// ============================================
// DB_RecipeProgram2 - Program 2
// Lines: 500
// CHUNKS: 5 x 100
// Generated by SpinningCam  [2026-09-29 00:03:31]
// !!! CONTINUOUS MOTION (CMD=2) - EXPERIMENTAL PLC ONLY !!!
// Load ONLY on the continuous-motion PLC build. A production PLC
// skips CMD=2 lines and jumps straight between the other points.
// T=0.045 s, corner tol=0.2 mm, F min=180, exact stop at >= 90 deg, stop slow-down=OFF
// CMD=2 lines: 385, exact corners: 39, slowed corners: 36 (+57 leaving), slowed stops: 0
// ============================================
//
// --- MAKINE AYARLARI ---
// Machine Origin  : X=0.0, Z=0.0
// Axis Direction  : X=NORMAL, Z=NORMAL
// Output Mode     : RADIUS
// G54 Offset      : X=0.0, Z=0.0
// Home            : X=-394.0, Z=-174.0
// Retract         : X=-10.0, Z=-10.0
//
// --- PARCA / BLANK ---
// Blank Radius    : 77.8 mm
// Blank Z Shift   : 0.0 mm
// Final Thickness : 0.8 mm
// Min Safety Gap  : 0.0 mm
//
// --- MANDREL POZISYON ---
// Mandrel Offset  : X=0.0, Z=0.0
// Mandrel Rot     : Rx=90.0, Ry=0.0, Rz=0.0
//
// --- OPERASYONLAR ---
// Op1: ROUGHING, 1 paso, T004, R=44.56mm, RPM=600.0, mm_min=900.0
// Op2: ROUGHING, 1 paso, T004, R=44.56mm, RPM=600.0, mm_min=900.0
// Op3: ROUGHING, 1 paso, T004, R=44.56mm, RPM=600.0, mm_min=900.0
// Op4: ROUGHING, 1 paso, T004, R=44.56mm, RPM=600.0, mm_min=900.0
// Op5: ROUGHING, 1 paso, T004, R=44.56mm, RPM=600.0, mm_min=900.0
// Op6: ROUGHING, 1 paso, T004, R=44.56mm, RPM=600.0, mm_min=800.0
// Op7: ROUGHING, 1 paso, T004, R=44.56mm, RPM=600.0, mm_min=800.0
// Op8: ROUGHING, 1 paso, T004, R=44.56mm, RPM=600.0, mm_min=800.0
// Op9: ROUGHING, 1 paso, T004, R=44.56mm, RPM=600.0, mm_min=800.0
// Op10: ROUGHING, 1 paso, T004, R=44.56mm, RPM=600.0, mm_min=800.0
// Op11: ROUGHING, 1 paso, T004, R=44.56mm, RPM=600.0, mm_min=800.0
// Op12: ROUGHING, 1 paso, T004, R=44.56mm, RPM=600.0, mm_min=800.0
// Op13: ROUGHING, 1 paso, T004, R=44.56mm, RPM=600.0, mm_min=1000.0
// Op14: ROUGHING, 1 paso, T004, R=44.56mm, RPM=600.0, mm_min=1000.0
// Op15: ROUGHING, 1 paso, T004, R=44.56mm, RPM=600.0, mm_min=1000.0
// Op16: ROUGHING, 1 paso, T004, R=44.56mm, RPM=600.0, mm_min=1000.0
// Op17: ROUGHING, 1 paso, T004, R=44.56mm, RPM=600.0, mm_min=1000.0
// Op18: ROUGHING, 1 paso, T004, R=44.56mm, RPM=600.0, mm_min=1000.0
// Op19: ROUGHING, 1 paso, T004, R=44.56mm, RPM=600.0, mm_min=1000.0
// Op20: ROUGHING, 1 paso, T004, R=44.56mm, RPM=600.0, mm_min=1000.0
// Op21: ROUGHING, 1 paso, T004, R=44.56mm, RPM=600.0, mm_min=1000.0
// Op22: ROUGHING, 1 paso, T004, R=44.56mm, RPM=600.0, mm_min=1000.0
// Op23: ROUGHING, 1 paso, T004, R=44.56mm, RPM=600.0, mm_min=1000.0
// Op24: ROUGHING, 1 paso, T004, R=44.56mm, RPM=600.0, mm_min=1000.0
// Op25: ROUGHING, 1 paso, T004, R=44.56mm, RPM=600.0, mm_min=1000.0
// Op26: ROUGHING, 1 paso, T004, R=44.56mm, RPM=600.0, mm_min=1000.0
// Op27: CUTTING, 1 paso, T006, R=20.0mm, RPM=500.0, mm_min=10.0
// Op28: ROUGHING, 1 paso, T004, R=44.56mm, RPM=600.0, mm_min=1000.0
// Op29: ROUGHING, 1 paso, T004, R=44.56mm, RPM=600.0, mm_min=1000.0
// Op30: ROUGHING, 1 paso, T004, R=44.56mm, RPM=600.0, mm_min=1000.0
// Op31: ROUGHING, 1 paso, T004, R=44.56mm, RPM=600.0, mm_min=1000.0
// Op32: ROUGHING, 1 paso, T004, R=44.56mm, RPM=600.0, mm_min=1000.0
// Op33: ROUGHING, 1 paso, T004, R=44.56mm, RPM=600.0, mm_min=1000.0
// Op34: ROUGHING, 1 paso, T004, R=44.56mm, RPM=600.0, mm_min=1000.0
// Op35: ROUGHING, 1 paso, T004, R=44.56mm, RPM=600.0, mm_min=1000.0
// Op36: ROUGHING, 1 paso, T004, R=44.56mm, RPM=600.0, mm_min=1500.0
// Op37: ROUGHING, 1 paso, T004, R=44.56mm, RPM=600.0, mm_min=1500.0
// Op38: ROUGHING, 1 paso, T004, R=44.56mm, RPM=600.0, mm_min=1500.0
// Op39: ROUGHING, 1 paso, T004, R=44.56mm, RPM=600.0, mm_min=1500.0
// Op40: ROUGHING, 1 paso, T004, R=44.56mm, RPM=600.0, mm_min=1500.0
// Op41: ROUGHING, 1 paso, T004, R=44.56mm, RPM=600.0, mm_min=1500.0
// Op42: ROUGHING, 1 paso, T004, R=44.56mm, RPM=600.0, mm_min=1500.0
// Op43: ROUGHING, 1 paso, T004, R=44.56mm, RPM=600.0, mm_min=1500.0
// Op44: ROUGHING, 1 paso, T004, R=44.56mm, RPM=600.0, mm_min=1500.0
// Op45: ROUGHING, 1 paso, T004, R=44.56mm, RPM=600.0, mm_min=1500.0
// Op46: ROUGHING, 1 paso, T004, R=44.56mm, RPM=600.0, mm_min=1500.0
// Op47: ROUGHING, 1 paso, T004, R=44.56mm, RPM=600.0, mm_min=1500.0
// Op48: ROUGHING, 1 paso, T004, R=44.56mm, RPM=600.0, mm_min=1500.0
// Op49: ROUGHING, 1 paso, T004, R=44.56mm, RPM=600.0, mm_min=1500.0
// Op50: ROUGHING, 1 paso, T004, R=44.56mm, RPM=600.0, mm_min=1500.0
// Op51: ROUGHING, 1 paso, T004, R=44.56mm, RPM=600.0, mm_min=1500.0
// Op52: ROUGHING, 1 paso, T004, R=44.56mm, RPM=600.0, mm_min=1500.0
// Op53: ROUGHING, 1 paso, T004, R=44.56mm, RPM=600.0, mm_min=1500.0
// Op54: ROUGHING, 1 paso, T004, R=44.56mm, RPM=600.0, mm_min=1500.0
// Op55: ROUGHING, 1 paso, T004, R=44.56mm, RPM=600.0, mm_min=1500.0
// Op56: ROUGHING, 1 paso, T004, R=44.56mm, RPM=600.0, mm_min=1500.0
// Op57: ROUGHING, 1 paso, T004, R=44.56mm, RPM=600.0, mm_min=1500.0
// Op58: ROUGHING, 1 paso, T004, R=44.56mm, RPM=600.0, mm_min=1500.0
// Op59: ROUGHING, 1 paso, T004, R=44.56mm, RPM=600.0, mm_min=1500.0
// Op60: ROUGHING, 1 paso, T004, R=44.56mm, RPM=800.0, mm_min=1500.0
// Op61: ROUGHING, 1 paso, T004, R=44.56mm, RPM=800.0, mm_min=800.0
// Op62: ROUGHING, 1 paso, T004, R=44.56mm, RPM=800.0, mm_min=800.0
// Op63: ROUGHING, 1 paso, T004, R=44.56mm, RPM=600.0, mm_min=1500.0
// Op64: ROUGHING, 1 paso, T004, R=44.56mm, RPM=600.0, mm_min=1500.0
// Op65: ROUGHING, 1 paso, T004, R=44.56mm, RPM=600.0, mm_min=1500.0
// Op66: ROUGHING, 1 paso, T004, R=44.56mm, RPM=600.0, mm_min=1500.0
// Op67: ROUGHING, 1 paso, T004, R=44.56mm, RPM=600.0, mm_min=1500.0
// Op68: ROUGHING, 1 paso, T004, R=44.56mm, RPM=600.0, mm_min=1500.0
// Op69: ROUGHING, 1 paso, T004, R=44.56mm, RPM=600.0, mm_min=1500.0
// Op70: ROUGHING, 1 paso, T004, R=44.56mm, RPM=600.0, mm_min=1500.0
// Op71: ROUGHING, 1 paso, T004, R=44.56mm, RPM=600.0, mm_min=1500.0
// Op72: ROUGHING, 1 paso, T004, R=44.56mm, RPM=600.0, mm_min=1000.0
// Op73: ROUGHING, 1 paso, T004, R=44.56mm, RPM=600.0, mm_min=1000.0
// Op74: ROUGHING, 1 paso, T004, R=44.56mm, RPM=600.0, mm_min=1000.0
// Op75: ROUGHING, 1 paso, T004, R=44.56mm, RPM=600.0, mm_min=1000.0
// Op76: ROUGHING, 1 paso, T004, R=44.56mm, RPM=600.0, mm_min=1500.0
// Op77: ROUGHING, 1 paso, T004, R=44.56mm, RPM=600.0, mm_min=1000.0
// Op78: ROUGHING, 1 paso, T004, R=44.56mm, RPM=600.0, mm_min=1000.0
// Op79: ROUGHING, 1 paso, T004, R=44.56mm, RPM=600.0, mm_min=1000.0
// Op80: ROUGHING, 1 paso, T004, R=44.56mm, RPM=600.0, mm_min=1000.0
// Op81: ROUGHING, 1 paso, T004, R=44.56mm, RPM=600.0, mm_min=1000.0
// Op82: ROUGHING, 1 paso, T004, R=44.56mm, RPM=600.0, mm_min=1000.0
// Op83: ROUGHING, 1 paso, T004, R=44.56mm, RPM=600.0, mm_min=1000.0
// Op84: ROUGHING, 1 paso, T004, R=44.56mm, RPM=600.0, mm_min=1000.0
// Op85: ROUGHING, 1 paso, T004, R=44.56mm, RPM=600.0, mm_min=1000.0
// Op86: ROUGHING, 1 paso, T004, R=44.56mm, RPM=600.0, mm_min=1000.0
// Op87: ROUGHING, 1 paso, T004, R=44.56mm, RPM=600.0, mm_min=1000.0
// Op88: ROUGHING, 1 paso, T004, R=44.56mm, RPM=600.0, mm_min=1000.0
// Op89: ROUGHING, 1 paso, T004, R=44.56mm, RPM=600.0, mm_min=1000.0
// Op90: ROUGHING, 1 paso, T004, R=44.56mm, RPM=600.0, mm_min=1000.0
// Op91: ROUGHING, 1 paso, T004, R=44.56mm, RPM=600.0, mm_min=1000.0
// Op92: ROUGHING, 1 paso, T004, R=44.56mm, RPM=600.0, mm_min=1000.0
// Op93: ROUGHING, 1 paso, T004, R=44.56mm, RPM=600.0, mm_min=1000.0
// Op94: ROUGHING, 1 paso, T004, R=44.56mm, RPM=600.0, mm_min=1000.0
// Op95: ROUGHING, 1 paso, T004, R=44.56mm, RPM=600.0, mm_min=1000.0
// Op96: ROUGHING, 1 paso, T004, R=44.56mm, RPM=600.0, mm_min=1000.0
// Op97: ROUGHING, 1 paso, T004, R=44.56mm, RPM=600.0, mm_min=1000.0
// Op98: ROUGHING, 1 paso, T004, R=44.56mm, RPM=600.0, mm_min=1000.0
// Op99: ROUGHING, 1 paso, T004, R=44.56mm, RPM=600.0, mm_min=1000.0
// Op100: ROUGHING, 1 paso, T004, R=44.56mm, RPM=600.0, mm_min=1000.0
// Op101: ROUGHING, 1 paso, T004, R=44.56mm, RPM=600.0, mm_min=1000.0
// Op102: ROUGHING, 1 paso, T004, R=44.56mm, RPM=600.0, mm_min=1000.0
// Op103: ROUGHING, 1 paso, T004, R=44.56mm, RPM=600.0, mm_min=1000.0
// Op104: ROUGHING, 1 paso, T004, R=44.56mm, RPM=600.0, mm_min=1000.0
// Op105: ROUGHING, 1 paso, T004, R=44.56mm, RPM=600.0, mm_min=1000.0
// Op106: ROUGHING, 1 paso, T004, R=44.56mm, RPM=600.0, mm_min=1000.0
// Op107: ROUGHING, 1 paso, T004, R=44.56mm, RPM=600.0, mm_min=1000.0
// Op108: ROUGHING, 1 paso, T004, R=44.56mm, RPM=600.0, mm_min=1000.0
// Op109: ROUGHING, 1 paso, T004, R=44.56mm, RPM=600.0, mm_min=1000.0
// Op110: ROUGHING, 1 paso, T004, R=44.56mm, RPM=600.0, mm_min=1000.0
// Op111: ROUGHING, 1 paso, T004, R=44.56mm, RPM=600.0, mm_min=1000.0
// Op112: ROUGHING, 1 paso, T004, R=44.56mm, RPM=600.0, mm_min=1000.0
// Op113: ROUGHING, 1 paso, T004, R=44.56mm, RPM=600.0, mm_min=1000.0
// Op114: ROUGHING, 1 paso, T004, R=44.56mm, RPM=600.0, mm_min=1000.0
// Op115: ROUGHING, 1 paso, T004, R=44.56mm, RPM=600.0, mm_min=1000.0
// Op116: ROUGHING, 1 paso, T004, R=44.56mm, RPM=600.0, mm_min=1000.0
// Op117: ROUGHING, 1 paso, T004, R=44.56mm, RPM=600.0, mm_min=1000.0
// Op118: ROUGHING, 1 paso, T004, R=44.56mm, RPM=600.0, mm_min=1000.0
// Op119: ROUGHING, 1 paso, T004, R=44.56mm, RPM=600.0, mm_min=1000.0
// Op120: ROUGHING, 1 paso, T004, R=44.56mm, RPM=600.0, mm_min=1000.0
// Op121: ROUGHING, 1 paso, T004, R=44.56mm, RPM=600.0, mm_min=1000.0
// Op122: ROUGHING, 1 paso, T004, R=44.56mm, RPM=600.0, mm_min=1000.0
// Op123: ROUGHING, 1 paso, T004, R=44.56mm, RPM=600.0, mm_min=1000.0
// Op124: ROUGHING, 1 paso, T004, R=44.56mm, RPM=600.0, mm_min=1000.0
// Op125: ROUGHING, 1 paso, T004, R=44.56mm, RPM=600.0, mm_min=1000.0
// Op126: ROUGHING, 1 paso, T004, R=44.56mm, RPM=600.0, mm_min=1000.0
// Op127: ROUGHING, 1 paso, T004, R=44.56mm, RPM=600.0, mm_min=1000.0
// Op128: ROUGHING, 1 paso, T004, R=44.56mm, RPM=600.0, mm_min=1000.0
// Op129: CUTTING, 1 paso, T006, R=20.0mm, RPM=500.0, mm_min=7.0
// Op130: ROUGHING, 1 paso, T004, R=44.56mm, RPM=600.0, mm_min=1000.0
// Op131: ROUGHING, 1 paso, T004, R=44.56mm, RPM=600.0, mm_min=1000.0
// Op132: ROUGHING, 1 paso, T004, R=44.56mm, RPM=600.0, mm_min=1000.0
// Op133: ROUGHING, 1 paso, T004, R=44.56mm, RPM=600.0, mm_min=1000.0
// Op134: ROUGHING, 1 paso, T004, R=44.56mm, RPM=600.0, mm_min=1000.0
// Op135: ROUGHING, 1 paso, T004, R=44.56mm, RPM=600.0, mm_min=1000.0
// Op136: ROUGHING, 1 paso, T004, R=44.56mm, RPM=600.0, mm_min=1000.0
// Op137: ROUGHING, 1 paso, T004, R=44.56mm, RPM=600.0, mm_min=400.0
// Op138: ROUGHING, 1 paso, T004, R=44.56mm, RPM=600.0, mm_min=400.0
// Op139: ROUGHING, 1 paso, T004, R=44.56mm, RPM=600.0, mm_min=400.0
// Op140: ROUGHING, 1 paso, T004, R=44.56mm, RPM=600.0, mm_min=1000.0
// Op141: ROUGHING, 1 paso, T004, R=44.56mm, RPM=600.0, mm_min=400.0
// Op142: ROUGHING, 1 paso, T004, R=44.56mm, RPM=600.0, mm_min=400.0
// Op143: ROUGHING, 1 paso, T004, R=44.56mm, RPM=600.0, mm_min=400.0
// Op144: ROUGHING, 1 paso, T004, R=44.56mm, RPM=600.0, mm_min=400.0
// Op145: ROUGHING, 1 paso, T004, R=44.56mm, RPM=600.0, mm_min=400.0
// Op146: ROUGHING, 1 paso, T004, R=44.56mm, RPM=600.0, mm_min=400.0
// Op147: ROUGHING, 1 paso, T004, R=44.56mm, RPM=600.0, mm_min=400.0
// Op148: ROUGHING, 1 paso, T004, R=44.56mm, RPM=600.0, mm_min=400.0
// Op149: ROUGHING, 1 paso, T004, R=44.56mm, RPM=600.0, mm_min=400.0
// Op150: ROUGHING, 1 paso, T004, R=44.56mm, RPM=600.0, mm_min=400.0
// Op151: ROUGHING, 1 paso, T004, R=44.56mm, RPM=600.0, mm_min=400.0
// Op152: ROUGHING, 1 paso, T004, R=44.56mm, RPM=600.0, mm_min=400.0
// Op153: ROUGHING, 1 paso, T004, R=44.56mm, RPM=600.0, mm_min=400.0
// Op154: ROUGHING, 1 paso, T004, R=44.56mm, RPM=600.0, mm_min=400.0
// Op155: ROUGHING, 1 paso, T004, R=44.56mm, RPM=600.0, mm_min=400.0
// Op156: ROUGHING, 1 paso, T004, R=44.56mm, RPM=600.0, mm_min=400.0
// Op157: ROUGHING, 1 paso, T004, R=44.56mm, RPM=600.0, mm_min=400.0
// Op158: ROUGHING, 1 paso, T004, R=44.56mm, RPM=600.0, mm_min=400.0
// Op159: ROUGHING, 1 paso, T004, R=44.56mm, RPM=600.0, mm_min=400.0
// Op160: ROUGHING, 1 paso, T004, R=44.56mm, RPM=600.0, mm_min=400.0
// Op161: ROUGHING, 1 paso, T004, R=44.56mm, RPM=600.0, mm_min=400.0
// Op162: ROUGHING, 1 paso, T004, R=44.56mm, RPM=600.0, mm_min=400.0
// Op163: ROUGHING, 1 paso, T004, R=44.56mm, RPM=600.0, mm_min=400.0
// Op164: ROUGHING, 1 paso, T004, R=44.56mm, RPM=600.0, mm_min=400.0
// Op165: ROUGHING, 1 paso, T004, R=44.56mm, RPM=600.0, mm_min=400.0
// Op166: ROUGHING, 1 paso, T004, R=44.56mm, RPM=600.0, mm_min=400.0
// Op167: ROUGHING, 1 paso, T004, R=44.56mm, RPM=800.0, mm_min=400.0
// Op168: ROUGHING, 1 paso, T004, R=44.56mm, RPM=800.0, mm_min=400.0
// Op169: ROUGHING, 1 paso, T004, R=44.56mm, RPM=800.0, mm_min=400.0
// Op170: ROUGHING, 1 paso, T004, R=44.56mm, RPM=800.0, mm_min=400.0
// Op171: ROUGHING, 1 paso, T004, R=44.56mm, RPM=800.0, mm_min=400.0
// Op172: ROUGHING, 1 paso, T004, R=44.56mm, RPM=800.0, mm_min=400.0
// Op173: ROUGHING, 1 paso, T004, R=44.56mm, RPM=800.0, mm_min=400.0
// Op174: ROUGHING, 1 paso, T004, R=44.56mm, RPM=800.0, mm_min=400.0
// Op175: ROUGHING, 1 paso, T004, R=44.56mm, RPM=800.0, mm_min=400.0
// Op176: ROUGHING, 1 paso, T004, R=44.56mm, RPM=800.0, mm_min=400.0
// Op177: ROUGHING, 1 paso, T004, R=44.56mm, RPM=800.0, mm_min=400.0
// Op178: ROUGHING, 1 paso, T004, R=44.56mm, RPM=800.0, mm_min=400.0
// Op179: ROUGHING, 1 paso, T004, R=44.56mm, RPM=800.0, mm_min=400.0
// Op180: ROUGHING, 1 paso, T004, R=44.56mm, RPM=800.0, mm_min=400.0
// Op181: ROUGHING, 1 paso, T004, R=44.56mm, RPM=800.0, mm_min=400.0
// Op182: ROUGHING, 1 paso, T004, R=44.56mm, RPM=800.0, mm_min=400.0
// Op183: ROUGHING, 1 paso, T004, R=44.56mm, RPM=800.0, mm_min=400.0
// ============================================

DATA_BLOCK "DB_RecipeProgram2"
{ S7_Optimized_Access := 'FALSE' }
VERSION : 0.2
UNLINKED
NON_RETAIN
    VAR
        Header : "RecipeHeader";
        Lines1 : Array[0..99] of "RecipeLine";  // global lines 0..99
        Lines2 : Array[0..99] of "RecipeLine";  // global lines 100..199
        Lines3 : Array[0..99] of "RecipeLine";  // global lines 200..299
        Lines4 : Array[0..99] of "RecipeLine";  // global lines 300..399
        Lines5 : Array[0..99] of "RecipeLine";  // global lines 400..499
    END_VAR
BEGIN
    // Header
    Header.sName := 'Program 2';
    Header.LineCount := 500;
    Header.Valid := TRUE;
    Header.PreScanned := FALSE;
    Header.MinX := 0.000;
    Header.MaxX := 273.391;
    Header.MinZ := 0.000;
    Header.MaxZ := 344.140;

    // --- Tool table (CAM-authored) ---
    Header.ProvidesToolConfig := TRUE;
    Header.ToolCount := 4;
    Header.AutoCalcAngles := FALSE;
    Header.ToolCode_List[1] := 4;
    Header.ToolCode_List[2] := 5;
    Header.ToolCode_List[3] := 6;
    Header.ToolCode_List[4] := 7;
    Header.ToolAngle_List[1] := 0.0;
    Header.ToolAngle_List[2] := 120.0;
    Header.ToolAngle_List[3] := 240.0;
    Header.ToolAngle_List[4] := 360.0;

    // --- Integrity ---
    // Order-sensitive sum over CMD+Param+F of lines 0..LineCount-1.
    // The PLC recomputes it after reassembling the chunks and refuses
    // to run on a mismatch (16#0316). X/Z are excluded on purpose:
    // float32-vs-float64 rounding would eventually cry wolf.
    Header.ProvidesChecksum := TRUE;
    Header.Checksum := 106433390;

    // Recipe Lines (500 total)

    // --- Lines1 (global lines 0..99) ---
    Lines1[0].X := 0.000; Lines1[0].Z := 0.000; Lines1[0].F := 0; Lines1[0].CMD := 40; Lines1[0].Param := 80; // Cylinder GOTO P80
    Lines1[1].X := 0.000; Lines1[1].Z := 0.000; Lines1[1].F := 0; Lines1[1].CMD := 10; Lines1[1].Param := 4; // Tool Change T4
    Lines1[2].X := 0.000; Lines1[2].Z := 0.000; Lines1[2].F := 0; Lines1[2].CMD := 20; Lines1[2].Param := 60; // Spindle ON 600 RPM
    Lines1[3].X := 0.000; Lines1[3].Z := 0.000; Lines1[3].F := 0; Lines1[3].CMD := 41; Lines1[3].Param := 1; // M41 (Clamp On) P1 [Op1 P1]
    Lines1[4].X := 272.912; Lines1[4].Z := 176.000; Lines1[4].F := 0; Lines1[4].CMD := 0; Lines1[4].Param := 0; // G0 Rapid [Op1 P1]
    Lines1[5].X := 272.901; Lines1[5].Z := 181.258; Lines1[5].F := 736; Lines1[5].CMD := 2; Lines1[5].Param := 0; // G1 Continuous [Op1 P1]
    Lines1[6].X := 272.111; Lines1[6].Z := 183.280; Lines1[6].F := 395; Lines1[6].CMD := 2; Lines1[6].Param := 0; // G1 Continuous [Op1 P1]
    Lines1[7].X := 270.164; Lines1[7].Z := 184.240; Lines1[7].F := 395; Lines1[7].CMD := 2; Lines1[7].Param := 0; // G1 Continuous [Op1 P1]
    Lines1[8].X := 178.498; Lines1[8].Z := 192.302; Lines1[8].F := 736; Lines1[8].CMD := 2; Lines1[8].Param := 0; // G1 Continuous [Op1 P1]
    Lines1[9].X := 173.498; Lines1[9].Z := 187.302; Lines1[9].F := 0; Lines1[9].CMD := 0; Lines1[9].Param := 0; // G0 Rapid [Op1 P1]
    Lines1[10].X := 173.498; Lines1[10].Z := 187.302; Lines1[10].F := 0; Lines1[10].CMD := 41; Lines1[10].Param := 2; // M41 (Clamp On) P2 [Op2 P1]
    Lines1[11].X := 273.001; Lines1[11].Z := 182.538; Lines1[11].F := 0; Lines1[11].CMD := 0; Lines1[11].Param := 0; // G0 Rapid [Op2 P1]
    Lines1[12].X := 272.998; Lines1[12].Z := 183.142; Lines1[12].F := 866; Lines1[12].CMD := 2; Lines1[12].Param := 0; // G1 Continuous [Op2 P1]
    Lines1[13].X := 272.418; Lines1[13].Z := 184.905; Lines1[13].F := 426; Lines1[13].CMD := 2; Lines1[13].Param := 0; // G1 Continuous [Op2 P1]
    Lines1[14].X := 270.650; Lines1[14].Z := 186.059; Lines1[14].F := 426; Lines1[14].CMD := 2; Lines1[14].Param := 0; // G1 Continuous [Op2 P1]
    Lines1[15].X := 180.388; Lines1[15].Z := 206.156; Lines1[15].F := 758; Lines1[15].CMD := 2; Lines1[15].Param := 0; // G1 Continuous [Op2 P1]
    Lines1[16].X := 272.995; Lines1[16].Z := 184.077; Lines1[16].F := 0; Lines1[16].CMD := 0; Lines1[16].Param := 0; // G0 Rapid [Op3 P1]
    Lines1[17].X := 272.992; Lines1[17].Z := 184.868; Lines1[17].F := 449; Lines1[17].CMD := 2; Lines1[17].Param := 0; // G1 Continuous [Op3 P1]
    Lines1[18].X := 270.873; Lines1[18].Z := 187.725; Lines1[18].F := 449; Lines1[18].CMD := 2; Lines1[18].Param := 0; // G1 Continuous [Op3 P1]
    Lines1[19].X := 182.286; Lines1[19].Z := 214.928; Lines1[19].F := 449; Lines1[19].CMD := 2; Lines1[19].Param := 0; // G1 Continuous [Op3 P1]
    Lines1[20].X := 273.006; Lines1[20].Z := 181.000; Lines1[20].F := 0; Lines1[20].CMD := 0; Lines1[20].Param := 0; // G0 Rapid [Op4 P1]
    Lines1[21].X := 272.984; Lines1[21].Z := 186.988; Lines1[21].F := 478; Lines1[21].CMD := 2; Lines1[21].Param := 0; // G1 Continuous [Op4 P1]
    Lines1[22].X := 271.113; Lines1[22].Z := 189.757; Lines1[22].F := 478; Lines1[22].CMD := 2; Lines1[22].Param := 0; // G1 Continuous [Op4 P1]
    Lines1[23].X := 185.053; Lines1[23].Z := 224.685; Lines1[23].F := 478; Lines1[23].CMD := 2; Lines1[23].Param := 0; // G1 Continuous [Op4 P1]
    Lines1[24].X := 273.006; Lines1[24].Z := 181.000; Lines1[24].F := 0; Lines1[24].CMD := 0; Lines1[24].Param := 0; // G0 Rapid [Op5 P1]
    Lines1[25].X := 272.980; Lines1[25].Z := 188.100; Lines1[25].F := 498; Lines1[25].CMD := 2; Lines1[25].Param := 0; // G1 Continuous [Op5 P1]
    Lines1[26].X := 271.253; Lines1[26].Z := 190.806; Lines1[26].F := 498; Lines1[26].CMD := 2; Lines1[26].Param := 0; // G1 Continuous [Op5 P1]
    Lines1[27].X := 187.038; Lines1[27].Z := 230.259; Lines1[27].F := 498; Lines1[27].CMD := 2; Lines1[27].Param := 0; // G1 Continuous [Op5 P1]
    Lines1[28].X := 273.106; Lines1[28].Z := 181.000; Lines1[28].F := 0; Lines1[28].CMD := 0; Lines1[28].Param := 0; // G0 Rapid [Op6 P1]
    Lines1[29].X := 273.076; Lines1[29].Z := 189.172; Lines1[29].F := 512; Lines1[29].CMD := 2; Lines1[29].Param := 0; // G1 Continuous [Op6 P1]
    Lines1[30].X := 271.442; Lines1[30].Z := 191.832; Lines1[30].F := 512; Lines1[30].CMD := 2; Lines1[30].Param := 0; // G1 Continuous [Op6 P1]
    Lines1[31].X := 188.492; Lines1[31].Z := 234.247; Lines1[31].F := 512; Lines1[31].CMD := 2; Lines1[31].Param := 0; // G1 Continuous [Op6 P1]
    Lines1[32].X := 273.106; Lines1[32].Z := 181.000; Lines1[32].F := 0; Lines1[32].CMD := 0; Lines1[32].Param := 0; // G0 Rapid [Op7 P1]
    Lines1[33].X := 273.072; Lines1[33].Z := 190.278; Lines1[33].F := 535; Lines1[33].CMD := 2; Lines1[33].Param := 0; // G1 Continuous [Op7 P1]
    Lines1[34].X := 271.576; Lines1[34].Z := 192.863; Lines1[34].F := 535; Lines1[34].CMD := 2; Lines1[34].Param := 0; // G1 Continuous [Op7 P1]
    Lines1[35].X := 190.869; Lines1[35].Z := 239.630; Lines1[35].F := 535; Lines1[35].CMD := 2; Lines1[35].Param := 0; // G1 Continuous [Op7 P1]
    Lines1[36].X := 273.106; Lines1[36].Z := 181.000; Lines1[36].F := 0; Lines1[36].CMD := 0; Lines1[36].Param := 0; // G0 Rapid [Op8 P1]
    Lines1[37].X := 273.068; Lines1[37].Z := 191.382; Lines1[37].F := 561; Lines1[37].CMD := 2; Lines1[37].Param := 0; // G1 Continuous [Op8 P1]
    Lines1[38].X := 271.707; Lines1[38].Z := 193.884; Lines1[38].F := 561; Lines1[38].CMD := 2; Lines1[38].Param := 0; // G1 Continuous [Op8 P1]
    Lines1[39].X := 193.471; Lines1[39].Z := 244.882; Lines1[39].F := 561; Lines1[39].CMD := 2; Lines1[39].Param := 0; // G1 Continuous [Op8 P1]
    Lines1[40].X := 273.206; Lines1[40].Z := 181.000; Lines1[40].F := 0; Lines1[40].CMD := 0; Lines1[40].Param := 0; // G0 Rapid [Op9 P1]
    Lines1[41].X := 273.164; Lines1[41].Z := 192.448; Lines1[41].F := 580; Lines1[41].CMD := 2; Lines1[41].Param := 0; // G1 Continuous [Op9 P1]
    Lines1[42].X := 271.888; Lines1[42].Z := 194.892; Lines1[42].F := 580; Lines1[42].CMD := 2; Lines1[42].Param := 0; // G1 Continuous [Op9 P1]
    Lines1[43].X := 234.859; Lines1[43].Z := 223.330; Lines1[43].F := 633; Lines1[43].CMD := 2; Lines1[43].Param := 0; // G1 Continuous [Op9 P1]
    Lines1[44].X := 195.326; Lines1[44].Z := 248.639; Lines1[44].F := 800; Lines1[44].CMD := 2; Lines1[44].Param := 0; // G1 Continuous [Op9 P1]
    Lines1[45].X := 273.206; Lines1[45].Z := 181.000; Lines1[45].F := 0; Lines1[45].CMD := 0; Lines1[45].Param := 0; // G0 Rapid [Op10 P1]
    Lines1[46].X := 273.164; Lines1[46].Z := 192.546; Lines1[46].F := 611; Lines1[46].CMD := 2; Lines1[46].Param := 0; // G1 Continuous [Op10 P1]
    Lines1[47].X := 272.014; Lines1[47].Z := 194.897; Lines1[47].F := 611; Lines1[47].CMD := 2; Lines1[47].Param := 0; // G1 Continuous [Op10 P1]
    Lines1[48].X := 236.288; Lines1[48].Z := 225.424; Lines1[48].F := 670; Lines1[48].CMD := 2; Lines1[48].Param := 0; // G1 Continuous [Op10 P1]
    Lines1[49].X := 198.293; Lines1[49].Z := 252.648; Lines1[49].F := 800; Lines1[49].CMD := 2; Lines1[49].Param := 0; // G1 Continuous [Op10 P1]
    Lines1[50].X := 273.206; Lines1[50].Z := 181.000; Lines1[50].F := 0; Lines1[50].CMD := 0; Lines1[50].Param := 0; // G0 Rapid [Op11 P1]
    Lines1[51].X := 273.164; Lines1[51].Z := 192.610; Lines1[51].F := 634; Lines1[51].CMD := 2; Lines1[51].Param := 0; // G1 Continuous [Op11 P1]
    Lines1[52].X := 272.095; Lines1[52].Z := 194.895; Lines1[52].F := 634; Lines1[52].CMD := 2; Lines1[52].Param := 0; // G1 Continuous [Op11 P1]
    Lines1[53].X := 255.662; Lines1[53].Z := 211.657; Lines1[53].F := 800; Lines1[53].CMD := 2; Lines1[53].Param := 0; // G1 Continuous [Op11 P1]
    Lines1[54].X := 238.268; Lines1[54].Z := 227.278; Lines1[54].F := 800; Lines1[54].CMD := 2; Lines1[54].Param := 0; // G1 Continuous [Op11 P1]
    Lines1[55].X := 219.711; Lines1[55].Z := 241.907; Lines1[55].F := 800; Lines1[55].CMD := 2; Lines1[55].Param := 0; // G1 Continuous [Op11 P1]
    Lines1[56].X := 200.385; Lines1[56].Z := 255.232; Lines1[56].F := 800; Lines1[56].CMD := 2; Lines1[56].Param := 0; // G1 Continuous [Op11 P1]
    Lines1[57].X := 273.206; Lines1[57].Z := 181.000; Lines1[57].F := 0; Lines1[57].CMD := 0; Lines1[57].Param := 0; // G0 Rapid [Op12 P1]
    Lines1[58].X := 273.164; Lines1[58].Z := 192.642; Lines1[58].F := 646; Lines1[58].CMD := 2; Lines1[58].Param := 0; // G1 Continuous [Op12 P1]
    Lines1[59].X := 272.135; Lines1[59].Z := 194.892; Lines1[59].F := 646; Lines1[59].CMD := 2; Lines1[59].Param := 0; // G1 Continuous [Op12 P1]
    Lines1[60].X := 256.846; Lines1[60].Z := 213.213; Lines1[60].F := 800; Lines1[60].CMD := 2; Lines1[60].Param := 0; // G1 Continuous [Op12 P1]
    Lines1[61].X := 240.086; Lines1[61].Z := 229.463; Lines1[61].F := 800; Lines1[61].CMD := 2; Lines1[61].Param := 0; // G1 Continuous [Op12 P1]
    Lines1[62].X := 221.493; Lines1[62].Z := 243.994; Lines1[62].F := 800; Lines1[62].CMD := 2; Lines1[62].Param := 0; // G1 Continuous [Op12 P1]
    Lines1[63].X := 201.465; Lines1[63].Z := 256.496; Lines1[63].F := 800; Lines1[63].CMD := 2; Lines1[63].Param := 0; // G1 Continuous [Op12 P1]
    Lines1[64].X := 273.206; Lines1[64].Z := 181.000; Lines1[64].F := 0; Lines1[64].CMD := 0; Lines1[64].Param := 0; // G0 Rapid [Op13 P1]
    Lines1[65].X := 273.163; Lines1[65].Z := 192.766; Lines1[65].F := 701; Lines1[65].CMD := 2; Lines1[65].Param := 0; // G1 Continuous [Op13 P1]
    Lines1[66].X := 272.288; Lines1[66].Z := 194.874; Lines1[66].F := 701; Lines1[66].CMD := 2; Lines1[66].Param := 0; // G1 Continuous [Op13 P1]
    Lines1[67].X := 258.825; Lines1[67].Z := 214.772; Lines1[67].F := 1000; Lines1[67].CMD := 2; Lines1[67].Param := 0; // G1 Continuous [Op13 P1]
    Lines1[68].X := 243.393; Lines1[68].Z := 232.353; Lines1[68].F := 1000; Lines1[68].CMD := 2; Lines1[68].Param := 0; // G1 Continuous [Op13 P1]
    Lines1[69].X := 225.658; Lines1[69].Z := 247.992; Lines1[69].F := 1000; Lines1[69].CMD := 2; Lines1[69].Param := 0; // G1 Continuous [Op13 P1]
    Lines1[70].X := 206.000; Lines1[70].Z := 261.359; Lines1[70].F := 1000; Lines1[70].CMD := 2; Lines1[70].Param := 0; // G1 Continuous [Op13 P1]
    Lines1[71].X := 273.206; Lines1[71].Z := 181.000; Lines1[71].F := 0; Lines1[71].CMD := 0; Lines1[71].Param := 0; // G0 Rapid [Op14 P1]
    Lines1[72].X := 273.163; Lines1[72].Z := 192.917; Lines1[72].F := 785; Lines1[72].CMD := 2; Lines1[72].Param := 0; // G1 Continuous [Op14 P1]
    Lines1[73].X := 272.464; Lines1[73].Z := 194.831; Lines1[73].F := 785; Lines1[73].CMD := 2; Lines1[73].Param := 0; // G1 Continuous [Op14 P1]
    Lines1[74].X := 260.797; Lines1[74].Z := 215.807; Lines1[74].F := 1000; Lines1[74].CMD := 2; Lines1[74].Param := 0; // G1 Continuous [Op14 P1]
    Lines1[75].X := 246.817; Lines1[75].Z := 234.848; Lines1[75].F := 1000; Lines1[75].CMD := 2; Lines1[75].Param := 0; // G1 Continuous [Op14 P1]
    Lines1[76].X := 230.709; Lines1[76].Z := 251.782; Lines1[76].F := 1000; Lines1[76].CMD := 2; Lines1[76].Param := 0; // G1 Continuous [Op14 P1]
    Lines1[77].X := 212.127; Lines1[77].Z := 266.973; Lines1[77].F := 1000; Lines1[77].CMD := 2; Lines1[77].Param := 0; // G1 Continuous [Op14 P1]
    Lines1[78].X := 273.206; Lines1[78].Z := 181.000; Lines1[78].F := 0; Lines1[78].CMD := 0; Lines1[78].Param := 0; // G0 Rapid [Op15 P1]
    Lines1[79].X := 273.162; Lines1[79].Z := 193.034; Lines1[79].F := 869; Lines1[79].CMD := 2; Lines1[79].Param := 0; // G1 Continuous [Op15 P1]
    Lines1[80].X := 272.592; Lines1[80].Z := 194.782; Lines1[80].F := 869; Lines1[80].CMD := 2; Lines1[80].Param := 0; // G1 Continuous [Op15 P1]
    Lines1[81].X := 262.089; Lines1[81].Z := 216.936; Lines1[81].F := 1000; Lines1[81].CMD := 2; Lines1[81].Param := 0; // G1 Continuous [Op15 P1]
    Lines1[82].X := 249.034; Lines1[82].Z := 237.552; Lines1[82].F := 1000; Lines1[82].CMD := 2; Lines1[82].Param := 0; // G1 Continuous [Op15 P1]
    Lines1[83].X := 233.696; Lines1[83].Z := 256.205; Lines1[83].F := 1000; Lines1[83].CMD := 2; Lines1[83].Param := 0; // G1 Continuous [Op15 P1]
    Lines1[84].X := 215.756; Lines1[84].Z := 273.284; Lines1[84].F := 1000; Lines1[84].CMD := 2; Lines1[84].Param := 0; // G1 Continuous [Op15 P1]
    Lines1[85].X := 273.206; Lines1[85].Z := 181.000; Lines1[85].F := 0; Lines1[85].CMD := 0; Lines1[85].Param := 0; // G0 Rapid [Op16 P1]
    Lines1[86].X := 273.162; Lines1[86].Z := 193.092; Lines1[86].F := 919; Lines1[86].CMD := 2; Lines1[86].Param := 0; // G1 Continuous [Op16 P1]
    Lines1[87].X := 272.652; Lines1[87].Z := 194.754; Lines1[87].F := 919; Lines1[87].CMD := 2; Lines1[87].Param := 0; // G1 Continuous [Op16 P1]
    Lines1[88].X := 264.161; Lines1[88].Z := 218.108; Lines1[88].F := 1000; Lines1[88].CMD := 2; Lines1[88].Param := 0; // G1 Continuous [Op16 P1]
    Lines1[89].X := 252.245; Lines1[89].Z := 239.462; Lines1[89].F := 1000; Lines1[89].CMD := 2; Lines1[89].Param := 0; // G1 Continuous [Op16 P1]
    Lines1[90].X := 237.149; Lines1[90].Z := 258.377; Lines1[90].F := 1000; Lines1[90].CMD := 2; Lines1[90].Param := 0; // G1 Continuous [Op16 P1]
    Lines1[91].X := 218.558; Lines1[91].Z := 275.246; Lines1[91].F := 1000; Lines1[91].CMD := 1; Lines1[91].Param := 0; // G1 Linear [Op16 P1]
    Lines1[92].X := 237.323; Lines1[92].Z := 258.191; Lines1[92].F := 1000; Lines1[92].CMD := 2; Lines1[92].Param := 0; // G1 Continuous [Op16 P1]
    Lines1[93].X := 252.664; Lines1[93].Z := 238.835; Lines1[93].F := 1000; Lines1[93].CMD := 2; Lines1[93].Param := 0; // G1 Continuous [Op16 P1]
    Lines1[94].X := 264.581; Lines1[94].Z := 217.179; Lines1[94].F := 1000; Lines1[94].CMD := 2; Lines1[94].Param := 0; // G1 Continuous [Op16 P1]
    Lines1[95].X := 273.162; Lines1[95].Z := 193.092; Lines1[95].F := 1000; Lines1[95].CMD := 2; Lines1[95].Param := 0; // G1 Continuous [Op16 P1]
    Lines1[96].X := 273.104; Lines1[96].Z := 181.000; Lines1[96].F := 0; Lines1[96].CMD := 0; Lines1[96].Param := 0; // G0 Rapid [Op17 P1]
    Lines1[97].X := 273.378; Lines1[97].Z := 188.527; Lines1[97].F := 1000; Lines1[97].CMD := 2; Lines1[97].Param := 0; // G1 Continuous [Op17 P1]
    Lines1[98].X := 272.487; Lines1[98].Z := 200.535; Lines1[98].F := 1000; Lines1[98].CMD := 2; Lines1[98].Param := 0; // G1 Continuous [Op17 P1]
    Lines1[99].X := 269.636; Lines1[99].Z := 212.563; Lines1[99].F := 1000; Lines1[99].CMD := 2; Lines1[99].Param := 0; // G1 Continuous [Op17 P1]

    // --- Lines2 (global lines 100..199) ---
    Lines2[0].X := 264.791; Lines2[0].Z := 224.689; Lines2[0].F := 1000; Lines2[0].CMD := 2; Lines2[0].Param := 0; // G1 Continuous [Op17 P1]
    Lines2[1].X := 258.145; Lines2[1].Z := 236.492; Lines2[1].F := 1000; Lines2[1].CMD := 2; Lines2[1].Param := 0; // G1 Continuous [Op17 P1]
    Lines2[2].X := 249.546; Lines2[2].Z := 248.191; Lines2[2].F := 1000; Lines2[2].CMD := 2; Lines2[2].Param := 0; // G1 Continuous [Op17 P1]
    Lines2[3].X := 239.464; Lines2[3].Z := 259.088; Lines2[3].F := 1000; Lines2[3].CMD := 2; Lines2[3].Param := 0; // G1 Continuous [Op17 P1]
    Lines2[4].X := 227.978; Lines2[4].Z := 269.090; Lines2[4].F := 1000; Lines2[4].CMD := 2; Lines2[4].Param := 0; // G1 Continuous [Op17 P1]
    Lines2[5].X := 215.593; Lines2[5].Z := 277.707; Lines2[5].F := 1000; Lines2[5].CMD := 2; Lines2[5].Param := 0; // G1 Continuous [Op17 P1]
    Lines2[6].X := 215.393; Lines2[6].Z := 277.707; Lines2[6].F := 0; Lines2[6].CMD := 0; Lines2[6].Param := 0; // G0 Rapid [Op17 P1]
    Lines2[7].X := 229.615; Lines2[7].Z := 267.632; Lines2[7].F := 1000; Lines2[7].CMD := 2; Lines2[7].Param := 0; // G1 Continuous [Op17 P1]
    Lines2[8].X := 242.446; Lines2[8].Z := 255.900; Lines2[8].F := 1000; Lines2[8].CMD := 2; Lines2[8].Param := 0; // G1 Continuous [Op17 P1]
    Lines2[9].X := 253.592; Lines2[9].Z := 242.773; Lines2[9].F := 1000; Lines2[9].CMD := 2; Lines2[9].Param := 0; // G1 Continuous [Op17 P1]
    Lines2[10].X := 262.327; Lines2[10].Z := 229.114; Lines2[10].F := 1000; Lines2[10].CMD := 1; Lines2[10].Param := 0; // G1 Linear [Op17 P1]
    Lines2[11].X := 253.873; Lines2[11].Z := 243.641; Lines2[11].F := 1000; Lines2[11].CMD := 2; Lines2[11].Param := 0; // G1 Continuous [Op18 P1]
    Lines2[12].X := 243.179; Lines2[12].Z := 257.644; Lines2[12].F := 1000; Lines2[12].CMD := 2; Lines2[12].Param := 0; // G1 Continuous [Op18 P1]
    Lines2[13].X := 230.798; Lines2[13].Z := 270.391; Lines2[13].F := 1000; Lines2[13].CMD := 2; Lines2[13].Param := 0; // G1 Continuous [Op18 P1]
    Lines2[14].X := 217.133; Lines2[14].Z := 281.504; Lines2[14].F := 1000; Lines2[14].CMD := 1; Lines2[14].Param := 0; // G1 Linear [Op18 P1]
    Lines2[15].X := 235.500; Lines2[15].Z := 265.895; Lines2[15].F := 1000; Lines2[15].CMD := 2; Lines2[15].Param := 0; // G1 Continuous [Op18 P1]
    Lines2[16].X := 251.025; Lines2[16].Z := 247.731; Lines2[16].F := 1000; Lines2[16].CMD := 2; Lines2[16].Param := 0; // G1 Continuous [Op18 P1]
    Lines2[17].X := 273.157; Lines2[17].Z := 181.000; Lines2[17].F := 0; Lines2[17].CMD := 0; Lines2[17].Param := 0; // G0 Rapid [Op19 P1]
    Lines2[18].X := 273.378; Lines2[18].Z := 188.273; Lines2[18].F := 1000; Lines2[18].CMD := 2; Lines2[18].Param := 0; // G1 Continuous [Op19 P1]
    Lines2[19].X := 272.550; Lines2[19].Z := 201.304; Lines2[19].F := 1000; Lines2[19].CMD := 2; Lines2[19].Param := 0; // G1 Continuous [Op19 P1]
    Lines2[20].X := 269.963; Lines2[20].Z := 214.198; Lines2[20].F := 1000; Lines2[20].CMD := 2; Lines2[20].Param := 0; // G1 Continuous [Op19 P1]
    Lines2[21].X := 265.577; Lines2[21].Z := 227.303; Lines2[21].F := 1000; Lines2[21].CMD := 2; Lines2[21].Param := 0; // G1 Continuous [Op19 P1]
    Lines2[22].X := 259.530; Lines2[22].Z := 240.201; Lines2[22].F := 1000; Lines2[22].CMD := 2; Lines2[22].Param := 0; // G1 Continuous [Op19 P1]
    Lines2[23].X := 251.806; Lines2[23].Z := 252.927; Lines2[23].F := 1000; Lines2[23].CMD := 2; Lines2[23].Param := 0; // G1 Continuous [Op19 P1]
    Lines2[24].X := 242.491; Lines2[24].Z := 265.231; Lines2[24].F := 1000; Lines2[24].CMD := 2; Lines2[24].Param := 0; // G1 Continuous [Op19 P1]
    Lines2[25].X := 231.907; Lines2[25].Z := 276.641; Lines2[25].F := 1000; Lines2[25].CMD := 2; Lines2[25].Param := 0; // G1 Continuous [Op19 P1]
    Lines2[26].X := 220.471; Lines2[26].Z := 286.742; Lines2[26].F := 1000; Lines2[26].CMD := 2; Lines2[26].Param := 0; // G1 Continuous [Op19 P1]
    Lines2[27].X := 220.271; Lines2[27].Z := 286.742; Lines2[27].F := 0; Lines2[27].CMD := 0; Lines2[27].Param := 0; // G0 Rapid [Op19 P1]
    Lines2[28].X := 233.901; Lines2[28].Z := 274.458; Lines2[28].F := 1000; Lines2[28].CMD := 2; Lines2[28].Param := 0; // G1 Continuous [Op19 P1]
    Lines2[29].X := 246.066; Lines2[29].Z := 260.552; Lines2[29].F := 1000; Lines2[29].CMD := 2; Lines2[29].Param := 0; // G1 Continuous [Op19 P1]
    Lines2[30].X := 256.379; Lines2[30].Z := 245.424; Lines2[30].F := 1000; Lines2[30].CMD := 2; Lines2[30].Param := 0; // G1 Continuous [Op19 P1]
    Lines2[31].X := 264.355; Lines2[31].Z := 229.767; Lines2[31].F := 1000; Lines2[31].CMD := 1; Lines2[31].Param := 0; // G1 Linear [Op19 P1]
    Lines2[32].X := 257.159; Lines2[32].Z := 245.114; Lines2[32].F := 1000; Lines2[32].CMD := 2; Lines2[32].Param := 0; // G1 Continuous [Op20 P1]
    Lines2[33].X := 247.934; Lines2[33].Z := 260.160; Lines2[33].F := 1000; Lines2[33].CMD := 2; Lines2[33].Param := 0; // G1 Continuous [Op20 P1]
    Lines2[34].X := 237.042; Lines2[34].Z := 274.255; Lines2[34].F := 1000; Lines2[34].CMD := 2; Lines2[34].Param := 0; // G1 Continuous [Op20 P1]
    Lines2[35].X := 224.733; Lines2[35].Z := 287.072; Lines2[35].F := 1000; Lines2[35].CMD := 1; Lines2[35].Param := 0; // G1 Linear [Op20 P1]
    Lines2[36].X := 241.468; Lines2[36].Z := 268.897; Lines2[36].F := 1000; Lines2[36].CMD := 2; Lines2[36].Param := 0; // G1 Continuous [Op20 P1]
    Lines2[37].X := 255.235; Lines2[37].Z := 248.577; Lines2[37].F := 1000; Lines2[37].CMD := 2; Lines2[37].Param := 0; // G1 Continuous [Op20 P1]
    Lines2[38].X := 273.155; Lines2[38].Z := 181.000; Lines2[38].F := 0; Lines2[38].CMD := 0; Lines2[38].Param := 0; // G0 Rapid [Op21 P1]
    Lines2[39].X := 273.377; Lines2[39].Z := 188.772; Lines2[39].F := 1000; Lines2[39].CMD := 2; Lines2[39].Param := 0; // G1 Continuous [Op21 P1]
    Lines2[40].X := 272.620; Lines2[40].Z := 202.062; Lines2[40].F := 1000; Lines2[40].CMD := 2; Lines2[40].Param := 0; // G1 Continuous [Op21 P1]
    Lines2[41].X := 270.277; Lines2[41].Z := 215.261; Lines2[41].F := 1000; Lines2[41].CMD := 2; Lines2[41].Param := 0; // G1 Continuous [Op21 P1]
    Lines2[42].X := 266.296; Lines2[42].Z := 228.732; Lines2[42].F := 1000; Lines2[42].CMD := 2; Lines2[42].Param := 0; // G1 Continuous [Op21 P1]
    Lines2[43].X := 260.669; Lines2[43].Z := 242.305; Lines2[43].F := 1000; Lines2[43].CMD := 2; Lines2[43].Param := 0; // G1 Continuous [Op21 P1]
    Lines2[44].X := 253.555; Lines2[44].Z := 255.558; Lines2[44].F := 1000; Lines2[44].CMD := 2; Lines2[44].Param := 0; // G1 Continuous [Op21 P1]
    Lines2[45].X := 245.069; Lines2[45].Z := 268.297; Lines2[45].F := 1000; Lines2[45].CMD := 2; Lines2[45].Param := 0; // G1 Continuous [Op21 P1]
    Lines2[46].X := 235.347; Lines2[46].Z := 280.310; Lines2[46].F := 1000; Lines2[46].CMD := 2; Lines2[46].Param := 0; // G1 Continuous [Op21 P1]
    Lines2[47].X := 224.726; Lines2[47].Z := 291.199; Lines2[47].F := 1000; Lines2[47].CMD := 2; Lines2[47].Param := 0; // G1 Continuous [Op21 P1]
    Lines2[48].X := 225.345; Lines2[48].Z := 275.927; Lines2[48].F := 0; Lines2[48].CMD := 0; Lines2[48].Param := 0; // G0 Rapid [Op22 P1]
    Lines2[49].X := 235.857; Lines2[49].Z := 267.484; Lines2[49].F := 1000; Lines2[49].CMD := 2; Lines2[49].Param := 0; // G1 Continuous [Op22 P1]
    Lines2[50].X := 245.453; Lines2[50].Z := 257.999; Lines2[50].F := 1000; Lines2[50].CMD := 2; Lines2[50].Param := 0; // G1 Continuous [Op22 P1]
    Lines2[51].X := 253.908; Lines2[51].Z := 247.702; Lines2[51].F := 1000; Lines2[51].CMD := 2; Lines2[51].Param := 0; // G1 Continuous [Op22 P1]
    Lines2[52].X := 260.898; Lines2[52].Z := 237.028; Lines2[52].F := 1000; Lines2[52].CMD := 2; Lines2[52].Param := 0; // G1 Continuous [Op22 P1]
    Lines2[53].X := 266.445; Lines2[53].Z := 225.966; Lines2[53].F := 1000; Lines2[53].CMD := 2; Lines2[53].Param := 0; // G1 Continuous [Op22 P1]
    Lines2[54].X := 270.351; Lines2[54].Z := 214.925; Lines2[54].F := 1000; Lines2[54].CMD := 2; Lines2[54].Param := 0; // G1 Continuous [Op22 P1]
    Lines2[55].X := 272.620; Lines2[55].Z := 204.069; Lines2[55].F := 1000; Lines2[55].CMD := 2; Lines2[55].Param := 0; // G1 Continuous [Op22 P1]
    Lines2[56].X := 273.363; Lines2[56].Z := 192.787; Lines2[56].F := 1000; Lines2[56].CMD := 2; Lines2[56].Param := 0; // G1 Continuous [Op22 P1]
    Lines2[57].X := 272.706; Lines2[57].Z := 181.000; Lines2[57].F := 1000; Lines2[57].CMD := 1; Lines2[57].Param := 0; // G1 Linear [Op22 P1]
    Lines2[58].X := 273.391; Lines2[58].Z := 181.000; Lines2[58].F := 1000; Lines2[58].CMD := 1; Lines2[58].Param := 0; // G1 Linear [Op23 P1]
    Lines2[59].X := 273.317; Lines2[59].Z := 203.231; Lines2[59].F := 1000; Lines2[59].CMD := 2; Lines2[59].Param := 0; // G1 Continuous [Op23 P1]
    Lines2[60].X := 272.942; Lines2[60].Z := 204.673; Lines2[60].F := 1000; Lines2[60].CMD := 2; Lines2[60].Param := 0; // G1 Continuous [Op23 P1]
    Lines2[61].X := 265.440; Lines2[61].Z := 230.646; Lines2[61].F := 1000; Lines2[61].CMD := 2; Lines2[61].Param := 0; // G1 Continuous [Op23 P1]
    Lines2[62].X := 254.420; Lines2[62].Z := 254.674; Lines2[62].F := 1000; Lines2[62].CMD := 2; Lines2[62].Param := 0; // G1 Continuous [Op23 P1]
    Lines2[63].X := 240.039; Lines2[63].Z := 276.555; Lines2[63].F := 1000; Lines2[63].CMD := 2; Lines2[63].Param := 0; // G1 Continuous [Op23 P1]
    Lines2[64].X := 222.020; Lines2[64].Z := 296.709; Lines2[64].F := 1000; Lines2[64].CMD := 1; Lines2[64].Param := 0; // G1 Linear [Op23 P1]
    Lines2[65].X := 238.475; Lines2[65].Z := 278.558; Lines2[65].F := 1000; Lines2[65].CMD := 2; Lines2[65].Param := 0; // G1 Continuous [Op23 P1]
    Lines2[66].X := 251.946; Lines2[66].Z := 258.991; Lines2[66].F := 1000; Lines2[66].CMD := 1; Lines2[66].Param := 0; // G1 Linear [Op23 P1]
    Lines2[67].X := 239.924; Lines2[67].Z := 278.409; Lines2[67].F := 1000; Lines2[67].CMD := 2; Lines2[67].Param := 0; // G1 Continuous [Op24 P1]
    Lines2[68].X := 225.658; Lines2[68].Z := 296.476; Lines2[68].F := 1000; Lines2[68].CMD := 1; Lines2[68].Param := 0; // G1 Linear [Op24 P1]
    Lines2[69].X := 236.341; Lines2[69].Z := 283.362; Lines2[69].F := 1000; Lines2[69].CMD := 2; Lines2[69].Param := 0; // G1 Continuous [Op24 P1]
    Lines2[70].X := 245.852; Lines2[70].Z := 269.448; Lines2[70].F := 1000; Lines2[70].CMD := 2; Lines2[70].Param := 0; // G1 Continuous [Op24 P1]
    Lines2[71].X := 254.088; Lines2[71].Z := 254.932; Lines2[71].F := 1000; Lines2[71].CMD := 2; Lines2[71].Param := 0; // G1 Continuous [Op24 P1]
    Lines2[72].X := 261.053; Lines2[72].Z := 239.761; Lines2[72].F := 1000; Lines2[72].CMD := 2; Lines2[72].Param := 0; // G1 Continuous [Op24 P1]
    Lines2[73].X := 266.452; Lines2[73].Z := 224.574; Lines2[73].F := 1000; Lines2[73].CMD := 2; Lines2[73].Param := 0; // G1 Continuous [Op24 P1]
    Lines2[74].X := 270.338; Lines2[74].Z := 209.300; Lines2[74].F := 1000; Lines2[74].CMD := 2; Lines2[74].Param := 0; // G1 Continuous [Op24 P1]
    Lines2[75].X := 272.653; Lines2[75].Z := 194.080; Lines2[75].F := 1000; Lines2[75].CMD := 2; Lines2[75].Param := 0; // G1 Continuous [Op24 P1]
    Lines2[76].X := 273.385; Lines2[76].Z := 179.043; Lines2[76].F := 1000; Lines2[76].CMD := 2; Lines2[76].Param := 0; // G1 Continuous [Op24 P1]
    Lines2[77].X := 273.022; Lines2[77].Z := 167.775; Lines2[77].F := 1000; Lines2[77].CMD := 2; Lines2[77].Param := 0; // G1 Continuous [Op24 P1]
    Lines2[78].X := 272.934; Lines2[78].Z := 181.000; Lines2[78].F := 0; Lines2[78].CMD := 0; Lines2[78].Param := 0; // G0 Rapid [Op25 P1]
    Lines2[79].X := 273.364; Lines2[79].Z := 192.276; Lines2[79].F := 1000; Lines2[79].CMD := 2; Lines2[79].Param := 0; // G1 Continuous [Op25 P1]
    Lines2[80].X := 272.654; Lines2[80].Z := 206.068; Lines2[80].F := 1000; Lines2[80].CMD := 2; Lines2[80].Param := 0; // G1 Continuous [Op25 P1]
    Lines2[81].X := 270.416; Lines2[81].Z := 219.773; Lines2[81].F := 1000; Lines2[81].CMD := 2; Lines2[81].Param := 0; // G1 Continuous [Op25 P1]
    Lines2[82].X := 266.578; Lines2[82].Z := 233.763; Lines2[82].F := 1000; Lines2[82].CMD := 2; Lines2[82].Param := 0; // G1 Continuous [Op25 P1]
    Lines2[83].X := 261.229; Lines2[83].Z := 247.642; Lines2[83].F := 1000; Lines2[83].CMD := 2; Lines2[83].Param := 0; // G1 Continuous [Op25 P1]
    Lines2[84].X := 254.448; Lines2[84].Z := 261.252; Lines2[84].F := 1000; Lines2[84].CMD := 2; Lines2[84].Param := 0; // G1 Continuous [Op25 P1]
    Lines2[85].X := 246.183; Lines2[85].Z := 274.631; Lines2[85].F := 1000; Lines2[85].CMD := 2; Lines2[85].Param := 0; // G1 Continuous [Op25 P1]
    Lines2[86].X := 236.652; Lines2[86].Z := 287.347; Lines2[86].F := 1000; Lines2[86].CMD := 2; Lines2[86].Param := 0; // G1 Continuous [Op25 P1]
    Lines2[87].X := 226.165; Lines2[87].Z := 299.007; Lines2[87].F := 1000; Lines2[87].CMD := 2; Lines2[87].Param := 0; // G1 Continuous [Op25 P1]
    Lines2[88].X := 229.789; Lines2[88].Z := 283.142; Lines2[88].F := 0; Lines2[88].CMD := 0; Lines2[88].Param := 0; // G0 Rapid [Op26 P1]
    Lines2[89].X := 239.436; Lines2[89].Z := 274.182; Lines2[89].F := 1000; Lines2[89].CMD := 2; Lines2[89].Param := 0; // G1 Continuous [Op26 P1]
    Lines2[90].X := 248.299; Lines2[90].Z := 264.192; Lines2[90].F := 1000; Lines2[90].CMD := 2; Lines2[90].Param := 0; // G1 Continuous [Op26 P1]
    Lines2[91].X := 256.017; Lines2[91].Z := 253.532; Lines2[91].F := 1000; Lines2[91].CMD := 2; Lines2[91].Param := 0; // G1 Continuous [Op26 P1]
    Lines2[92].X := 262.328; Lines2[92].Z := 242.612; Lines2[92].F := 1000; Lines2[92].CMD := 2; Lines2[92].Param := 0; // G1 Continuous [Op26 P1]
    Lines2[93].X := 267.192; Lines2[93].Z := 231.628; Lines2[93].F := 1000; Lines2[93].CMD := 2; Lines2[93].Param := 0; // G1 Continuous [Op26 P1]
    Lines2[94].X := 270.665; Lines2[94].Z := 220.497; Lines2[94].F := 1000; Lines2[94].CMD := 2; Lines2[94].Param := 0; // G1 Continuous [Op26 P1]
    Lines2[95].X := 272.687; Lines2[95].Z := 209.341; Lines2[95].F := 1000; Lines2[95].CMD := 2; Lines2[95].Param := 0; // G1 Continuous [Op26 P1]
    Lines2[96].X := 273.345; Lines2[96].Z := 197.787; Lines2[96].F := 1000; Lines2[96].CMD := 2; Lines2[96].Param := 0; // G1 Continuous [Op26 P1]
    Lines2[97].X := 272.130; Lines2[97].Z := 181.000; Lines2[97].F := 1000; Lines2[97].CMD := 2; Lines2[97].Param := 0; // G1 Continuous [Op26 P1]
    Lines2[98].X := 272.130; Lines2[98].Z := 181.000; Lines2[98].F := 0; Lines2[98].CMD := 0; Lines2[98].Param := 0; // G0 Rapid [Op26 P1]
    Lines2[99].X := 222.130; Lines2[99].Z := 181.000; Lines2[99].F := 0; Lines2[99].CMD := 0; Lines2[99].Param := 0; // G0 Rapid [Op26 P1]

    // --- Lines3 (global lines 200..299) ---
    Lines3[0].X := 222.130; Lines3[0].Z := 181.000; Lines3[0].F := 0; Lines3[0].CMD := 20; Lines3[0].Param := 50; // Spindle ON 500 RPM [Op26 P1]
    Lines3[1].X := 222.130; Lines3[1].Z := 181.000; Lines3[1].F := 0; Lines3[1].CMD := 10; Lines3[1].Param := 6; // Tool Change T6 [Op26 P1]
    Lines3[2].X := 219.000; Lines3[2].Z := 304.000; Lines3[2].F := 0; Lines3[2].CMD := 0; Lines3[2].Param := 0; // G0 Rapid [Op27 P1]
    Lines3[3].X := 227.000; Lines3[3].Z := 304.000; Lines3[3].F := 10; Lines3[3].CMD := 2; Lines3[3].Param := 0; // G1 Continuous [Op27 P1]
    Lines3[4].X := 177.000; Lines3[4].Z := 304.000; Lines3[4].F := 0; Lines3[4].CMD := 0; Lines3[4].Param := 0; // G0 Rapid [Op27 P1]
    Lines3[5].X := 177.000; Lines3[5].Z := 0.000; Lines3[5].F := 0; Lines3[5].CMD := 0; Lines3[5].Param := 0; // G0 Rapid [Op27 P1]
    Lines3[6].X := 0.000; Lines3[6].Z := 0.000; Lines3[6].F := 0; Lines3[6].CMD := 0; Lines3[6].Param := 0; // G0 Rapid [Op27 P1]
    Lines3[7].X := 0.000; Lines3[7].Z := 0.000; Lines3[7].F := 0; Lines3[7].CMD := 20; Lines3[7].Param := 60; // Spindle ON 600 RPM [Op27 P1]
    Lines3[8].X := 0.000; Lines3[8].Z := 0.000; Lines3[8].F := 0; Lines3[8].CMD := 10; Lines3[8].Param := 4; // Tool Change T4 [Op27 P1]
    Lines3[9].X := 272.415; Lines3[9].Z := 181.000; Lines3[9].F := 0; Lines3[9].CMD := 0; Lines3[9].Param := 0; // G0 Rapid [Op28 P1]
    Lines3[10].X := 273.345; Lines3[10].Z := 197.544; Lines3[10].F := 1000; Lines3[10].CMD := 2; Lines3[10].Param := 0; // G1 Continuous [Op28 P1]
    Lines3[11].X := 272.594; Lines3[11].Z := 211.604; Lines3[11].F := 1000; Lines3[11].CMD := 2; Lines3[11].Param := 0; // G1 Continuous [Op28 P1]
    Lines3[12].X := 270.331; Lines3[12].Z := 225.038; Lines3[12].F := 1000; Lines3[12].CMD := 2; Lines3[12].Param := 0; // G1 Continuous [Op28 P1]
    Lines3[13].X := 266.434; Lines3[13].Z := 238.719; Lines3[13].F := 1000; Lines3[13].CMD := 2; Lines3[13].Param := 0; // G1 Continuous [Op28 P1]
    Lines3[14].X := 260.893; Lines3[14].Z := 252.489; Lines3[14].F := 1000; Lines3[14].CMD := 2; Lines3[14].Param := 0; // G1 Continuous [Op28 P1]
    Lines3[15].X := 253.858; Lines3[15].Z := 265.944; Lines3[15].F := 1000; Lines3[15].CMD := 2; Lines3[15].Param := 0; // G1 Continuous [Op28 P1]
    Lines3[16].X := 245.288; Lines3[16].Z := 279.117; Lines3[16].F := 1000; Lines3[16].CMD := 2; Lines3[16].Param := 0; // G1 Continuous [Op28 P1]
    Lines3[17].X := 235.426; Lines3[17].Z := 291.579; Lines3[17].F := 1000; Lines3[17].CMD := 2; Lines3[17].Param := 0; // G1 Continuous [Op28 P1]
    Lines3[18].X := 224.610; Lines3[18].Z := 302.942; Lines3[18].F := 1000; Lines3[18].CMD := 1; Lines3[18].Param := 0; // G1 Linear [Op28 P1]
    Lines3[19].X := 235.259; Lines3[19].Z := 291.772; Lines3[19].F := 1000; Lines3[19].CMD := 2; Lines3[19].Param := 0; // G1 Continuous [Op28 P1]
    Lines3[20].X := 244.836; Lines3[20].Z := 279.743; Lines3[20].F := 1000; Lines3[20].CMD := 2; Lines3[20].Param := 0; // G1 Continuous [Op28 P1]
    Lines3[21].X := 253.202; Lines3[21].Z := 267.054; Lines3[21].F := 1000; Lines3[21].CMD := 2; Lines3[21].Param := 0; // G1 Continuous [Op28 P1]
    Lines3[22].X := 260.204; Lines3[22].Z := 253.958; Lines3[22].F := 1000; Lines3[22].CMD := 1; Lines3[22].Param := 0; // G1 Linear [Op28 P1]
    Lines3[23].X := 253.353; Lines3[23].Z := 267.713; Lines3[23].F := 1000; Lines3[23].CMD := 2; Lines3[23].Param := 0; // G1 Continuous [Op29 P1]
    Lines3[24].X := 245.192; Lines3[24].Z := 281.073; Lines3[24].F := 1000; Lines3[24].CMD := 2; Lines3[24].Param := 0; // G1 Continuous [Op29 P1]
    Lines3[25].X := 235.988; Lines3[25].Z := 293.639; Lines3[25].F := 1000; Lines3[25].CMD := 2; Lines3[25].Param := 0; // G1 Continuous [Op29 P1]
    Lines3[26].X := 225.720; Lines3[26].Z := 305.457; Lines3[26].F := 1000; Lines3[26].CMD := 1; Lines3[26].Param := 0; // G1 Linear [Op29 P1]
    Lines3[27].X := 237.406; Lines3[27].Z := 291.840; Lines3[27].F := 1000; Lines3[27].CMD := 2; Lines3[27].Param := 0; // G1 Continuous [Op29 P1]
    Lines3[28].X := 247.715; Lines3[28].Z := 277.207; Lines3[28].F := 1000; Lines3[28].CMD := 2; Lines3[28].Param := 0; // G1 Continuous [Op29 P1]
    Lines3[29].X := 256.478; Lines3[29].Z := 261.811; Lines3[29].F := 1000; Lines3[29].CMD := 2; Lines3[29].Param := 0; // G1 Continuous [Op29 P1]
    Lines3[30].X := 263.428; Lines3[30].Z := 246.178; Lines3[30].F := 1000; Lines3[30].CMD := 2; Lines3[30].Param := 0; // G1 Continuous [Op29 P1]
    Lines3[31].X := 272.550; Lines3[31].Z := 181.000; Lines3[31].F := 0; Lines3[31].CMD := 0; Lines3[31].Param := 0; // G0 Rapid [Op30 P1]
    Lines3[32].X := 273.346; Lines3[32].Z := 197.274; Lines3[32].F := 1000; Lines3[32].CMD := 2; Lines3[32].Param := 0; // G1 Continuous [Op30 P1]
    Lines3[33].X := 272.691; Lines3[33].Z := 211.571; Lines3[33].F := 1000; Lines3[33].CMD := 2; Lines3[33].Param := 0; // G1 Continuous [Op30 P1]
    Lines3[34].X := 270.722; Lines3[34].Z := 225.291; Lines3[34].F := 1000; Lines3[34].CMD := 2; Lines3[34].Param := 0; // G1 Continuous [Op30 P1]
    Lines3[35].X := 267.330; Lines3[35].Z := 239.330; Lines3[35].F := 1000; Lines3[35].CMD := 2; Lines3[35].Param := 0; // G1 Continuous [Op30 P1]
    Lines3[36].X := 262.575; Lines3[36].Z := 253.317; Lines3[36].F := 1000; Lines3[36].CMD := 2; Lines3[36].Param := 0; // G1 Continuous [Op30 P1]
    Lines3[37].X := 256.392; Lines3[37].Z := 267.350; Lines3[37].F := 1000; Lines3[37].CMD := 2; Lines3[37].Param := 0; // G1 Continuous [Op30 P1]
    Lines3[38].X := 249.049; Lines3[38].Z := 280.814; Lines3[38].F := 1000; Lines3[38].CMD := 2; Lines3[38].Param := 0; // G1 Continuous [Op30 P1]
    Lines3[39].X := 231.061; Lines3[39].Z := 305.913; Lines3[39].F := 1000; Lines3[39].CMD := 2; Lines3[39].Param := 0; // G1 Continuous [Op30 P1]
    Lines3[40].X := 223.990; Lines3[40].Z := 295.927; Lines3[40].F := 0; Lines3[40].CMD := 0; Lines3[40].Param := 0; // G0 Rapid [Op31 P1]
    Lines3[41].X := 235.026; Lines3[41].Z := 286.228; Lines3[41].F := 1000; Lines3[41].CMD := 2; Lines3[41].Param := 0; // G1 Continuous [Op31 P1]
    Lines3[42].X := 245.023; Lines3[42].Z := 275.525; Lines3[42].F := 1000; Lines3[42].CMD := 2; Lines3[42].Param := 0; // G1 Continuous [Op31 P1]
    Lines3[43].X := 253.765; Lines3[43].Z := 264.025; Lines3[43].F := 1000; Lines3[43].CMD := 2; Lines3[43].Param := 0; // G1 Continuous [Op31 P1]
    Lines3[44].X := 260.944; Lines3[44].Z := 252.145; Lines3[44].F := 1000; Lines3[44].CMD := 2; Lines3[44].Param := 0; // G1 Continuous [Op31 P1]
    Lines3[45].X := 266.483; Lines3[45].Z := 240.091; Lines3[45].F := 1000; Lines3[45].CMD := 2; Lines3[45].Param := 0; // G1 Continuous [Op31 P1]
    Lines3[46].X := 270.347; Lines3[46].Z := 228.042; Lines3[46].F := 1000; Lines3[46].CMD := 2; Lines3[46].Param := 0; // G1 Continuous [Op31 P1]
    Lines3[47].X := 272.584; Lines3[47].Z := 215.898; Lines3[47].F := 1000; Lines3[47].CMD := 2; Lines3[47].Param := 0; // G1 Continuous [Op31 P1]
    Lines3[48].X := 273.334; Lines3[48].Z := 203.063; Lines3[48].F := 1000; Lines3[48].CMD := 2; Lines3[48].Param := 0; // G1 Continuous [Op31 P1]
    Lines3[49].X := 271.416; Lines3[49].Z := 181.000; Lines3[49].F := 1000; Lines3[49].CMD := 1; Lines3[49].Param := 0; // G1 Linear [Op31 P1]
    Lines3[50].X := 271.919; Lines3[50].Z := 181.000; Lines3[50].F := 1000; Lines3[50].CMD := 1; Lines3[50].Param := 0; // G1 Linear [Op32 P1]
    Lines3[51].X := 273.335; Lines3[51].Z := 202.537; Lines3[51].F := 1000; Lines3[51].CMD := 2; Lines3[51].Param := 0; // G1 Continuous [Op32 P1]
    Lines3[52].X := 272.724; Lines3[52].Z := 216.104; Lines3[52].F := 1000; Lines3[52].CMD := 2; Lines3[52].Param := 0; // G1 Continuous [Op32 P1]
    Lines3[53].X := 270.870; Lines3[53].Z := 229.329; Lines3[53].F := 1000; Lines3[53].CMD := 2; Lines3[53].Param := 0; // G1 Continuous [Op32 P1]
    Lines3[54].X := 267.684; Lines3[54].Z := 242.612; Lines3[54].F := 1000; Lines3[54].CMD := 2; Lines3[54].Param := 0; // G1 Continuous [Op32 P1]
    Lines3[55].X := 263.192; Lines3[55].Z := 255.843; Lines3[55].F := 1000; Lines3[55].CMD := 2; Lines3[55].Param := 0; // G1 Continuous [Op32 P1]
    Lines3[56].X := 250.347; Lines3[56].Z := 281.884; Lines3[56].F := 1000; Lines3[56].CMD := 2; Lines3[56].Param := 0; // G1 Continuous [Op32 P1]
    Lines3[57].X := 232.895; Lines3[57].Z := 306.090; Lines3[57].F := 1000; Lines3[57].CMD := 1; Lines3[57].Param := 0; // G1 Linear [Op32 P1]
    Lines3[58].X := 242.231; Lines3[58].Z := 294.191; Lines3[58].F := 1000; Lines3[58].CMD := 2; Lines3[58].Param := 0; // G1 Continuous [Op32 P1]
    Lines3[59].X := 250.609; Lines3[59].Z := 281.447; Lines3[59].F := 1000; Lines3[59].CMD := 2; Lines3[59].Param := 0; // G1 Continuous [Op32 P1]
    Lines3[60].X := 257.775; Lines3[60].Z := 268.217; Lines3[60].F := 1000; Lines3[60].CMD := 2; Lines3[60].Param := 0; // G1 Continuous [Op32 P1]
    Lines3[61].X := 263.618; Lines3[61].Z := 254.737; Lines3[61].F := 1000; Lines3[61].CMD := 1; Lines3[61].Param := 0; // G1 Linear [Op32 P1]
    Lines3[62].X := 251.632; Lines3[62].Z := 282.331; Lines3[62].F := 1000; Lines3[62].CMD := 2; Lines3[62].Param := 0; // G1 Continuous [Op33 P1]
    Lines3[63].X := 235.569; Lines3[63].Z := 308.041; Lines3[63].F := 1000; Lines3[63].CMD := 1; Lines3[63].Param := 0; // G1 Linear [Op33 P1]
    Lines3[64].X := 251.869; Lines3[64].Z := 281.881; Lines3[64].F := 1000; Lines3[64].CMD := 2; Lines3[64].Param := 0; // G1 Continuous [Op33 P1]
    Lines3[65].X := 263.839; Lines3[65].Z := 254.095; Lines3[65].F := 1000; Lines3[65].CMD := 2; Lines3[65].Param := 0; // G1 Continuous [Op33 P1]
    Lines3[66].X := 271.025; Lines3[66].Z := 225.874; Lines3[66].F := 1000; Lines3[66].CMD := 2; Lines3[66].Param := 0; // G1 Continuous [Op33 P1]
    Lines3[67].X := 273.343; Lines3[67].Z := 197.537; Lines3[67].F := 1000; Lines3[67].CMD := 2; Lines3[67].Param := 0; // G1 Continuous [Op33 P1]
    Lines3[68].X := 272.146; Lines3[68].Z := 176.229; Lines3[68].F := 1000; Lines3[68].CMD := 1; Lines3[68].Param := 0; // G1 Linear [Op33 P1]
    Lines3[69].X := 273.342; Lines3[69].Z := 198.610; Lines3[69].F := 1000; Lines3[69].CMD := 2; Lines3[69].Param := 0; // G1 Continuous [Op34 P1]
    Lines3[70].X := 271.189; Lines3[70].Z := 227.191; Lines3[70].F := 1000; Lines3[70].CMD := 2; Lines3[70].Param := 0; // G1 Continuous [Op34 P1]
    Lines3[71].X := 264.640; Lines3[71].Z := 255.520; Lines3[71].F := 1000; Lines3[71].CMD := 2; Lines3[71].Param := 0; // G1 Continuous [Op34 P1]
    Lines3[72].X := 253.695; Lines3[72].Z := 283.639; Lines3[72].F := 1000; Lines3[72].CMD := 2; Lines3[72].Param := 0; // G1 Continuous [Op34 P1]
    Lines3[73].X := 238.799; Lines3[73].Z := 310.271; Lines3[73].F := 1000; Lines3[73].CMD := 1; Lines3[73].Param := 0; // G1 Linear [Op34 P1]
    Lines3[74].X := 253.695; Lines3[74].Z := 283.639; Lines3[74].F := 1000; Lines3[74].CMD := 2; Lines3[74].Param := 0; // G1 Continuous [Op34 P1]
    Lines3[75].X := 264.640; Lines3[75].Z := 255.520; Lines3[75].F := 1000; Lines3[75].CMD := 2; Lines3[75].Param := 0; // G1 Continuous [Op34 P1]
    Lines3[76].X := 271.189; Lines3[76].Z := 227.191; Lines3[76].F := 1000; Lines3[76].CMD := 2; Lines3[76].Param := 0; // G1 Continuous [Op34 P1]
    Lines3[77].X := 273.342; Lines3[77].Z := 198.610; Lines3[77].F := 1000; Lines3[77].CMD := 2; Lines3[77].Param := 0; // G1 Continuous [Op34 P1]
    Lines3[78].X := 272.255; Lines3[78].Z := 177.312; Lines3[78].F := 1000; Lines3[78].CMD := 2; Lines3[78].Param := 0; // G1 Continuous [Op34 P1]
    Lines3[79].X := 225.740; Lines3[79].Z := 301.695; Lines3[79].F := 0; Lines3[79].CMD := 0; Lines3[79].Param := 0; // G0 Rapid [Op35 P1]
    Lines3[80].X := 236.539; Lines3[80].Z := 291.770; Lines3[80].F := 1000; Lines3[80].CMD := 2; Lines3[80].Param := 0; // G1 Continuous [Op35 P1]
    Lines3[81].X := 246.275; Lines3[81].Z := 280.910; Lines3[81].F := 1000; Lines3[81].CMD := 2; Lines3[81].Param := 0; // G1 Continuous [Op35 P1]
    Lines3[82].X := 254.603; Lines3[82].Z := 269.518; Lines3[82].F := 1000; Lines3[82].CMD := 2; Lines3[82].Param := 0; // G1 Continuous [Op35 P1]
    Lines3[83].X := 261.537; Lines3[83].Z := 257.579; Lines3[83].F := 1000; Lines3[83].CMD := 2; Lines3[83].Param := 0; // G1 Continuous [Op35 P1]
    Lines3[84].X := 266.759; Lines3[84].Z := 245.719; Lines3[84].F := 1000; Lines3[84].CMD := 2; Lines3[84].Param := 0; // G1 Continuous [Op35 P1]
    Lines3[85].X := 270.446; Lines3[85].Z := 233.636; Lines3[85].F := 1000; Lines3[85].CMD := 2; Lines3[85].Param := 0; // G1 Continuous [Op35 P1]
    Lines3[86].X := 272.600; Lines3[86].Z := 221.207; Lines3[86].F := 1000; Lines3[86].CMD := 2; Lines3[86].Param := 0; // G1 Continuous [Op35 P1]
    Lines3[87].X := 273.317; Lines3[87].Z := 208.083; Lines3[87].F := 1000; Lines3[87].CMD := 2; Lines3[87].Param := 0; // G1 Continuous [Op35 P1]
    Lines3[88].X := 272.613; Lines3[88].Z := 194.693; Lines3[88].F := 1000; Lines3[88].CMD := 2; Lines3[88].Param := 0; // G1 Continuous [Op35 P1]
    Lines3[89].X := 270.536; Lines3[89].Z := 181.000; Lines3[89].F := 1000; Lines3[89].CMD := 1; Lines3[89].Param := 0; // G1 Linear [Op35 P1]
    Lines3[90].X := 271.713; Lines3[90].Z := 181.000; Lines3[90].F := 1000; Lines3[90].CMD := 1; Lines3[90].Param := 0; // G1 Linear [Op36 P1]
    Lines3[91].X := 273.319; Lines3[91].Z := 207.305; Lines3[91].F := 1500; Lines3[91].CMD := 2; Lines3[91].Param := 0; // G1 Continuous [Op36 P1]
    Lines3[92].X := 271.268; Lines3[92].Z := 235.902; Lines3[92].F := 1500; Lines3[92].CMD := 2; Lines3[92].Param := 0; // G1 Continuous [Op36 P1]
    Lines3[93].X := 264.960; Lines3[93].Z := 264.238; Lines3[93].F := 1500; Lines3[93].CMD := 2; Lines3[93].Param := 0; // G1 Continuous [Op36 P1]
    Lines3[94].X := 254.443; Lines3[94].Z := 292.178; Lines3[94].F := 1500; Lines3[94].CMD := 2; Lines3[94].Param := 0; // G1 Continuous [Op36 P1]
    Lines3[95].X := 239.952; Lines3[95].Z := 318.992; Lines3[95].F := 1500; Lines3[95].CMD := 1; Lines3[95].Param := 0; // G1 Linear [Op36 P1]
    Lines3[96].X := 248.760; Lines3[96].Z := 303.744; Lines3[96].F := 1500; Lines3[96].CMD := 2; Lines3[96].Param := 0; // G1 Continuous [Op36 P1]
    Lines3[97].X := 256.291; Lines3[97].Z := 288.015; Lines3[97].F := 1500; Lines3[97].CMD := 2; Lines3[97].Param := 0; // G1 Continuous [Op36 P1]
    Lines3[98].X := 262.491; Lines3[98].Z := 271.954; Lines3[98].F := 1500; Lines3[98].CMD := 2; Lines3[98].Param := 0; // G1 Continuous [Op36 P1]
    Lines3[99].X := 267.379; Lines3[99].Z := 255.445; Lines3[99].F := 1500; Lines3[99].CMD := 1; Lines3[99].Param := 0; // G1 Linear [Op36 P1]

    // --- Lines4 (global lines 300..399) ---
    Lines4[0].X := 257.701; Lines4[0].Z := 289.812; Lines4[0].F := 1500; Lines4[0].CMD := 2; Lines4[0].Param := 0; // G1 Continuous [Op37 P1]
    Lines4[1].X := 243.764; Lines4[1].Z := 322.929; Lines4[1].F := 1500; Lines4[1].CMD := 1; Lines4[1].Param := 0; // G1 Linear [Op37 P1]
    Lines4[2].X := 251.956; Lines4[2].Z := 304.869; Lines4[2].F := 1500; Lines4[2].CMD := 2; Lines4[2].Param := 0; // G1 Continuous [Op37 P1]
    Lines4[3].X := 258.928; Lines4[3].Z := 286.235; Lines4[3].F := 1500; Lines4[3].CMD := 2; Lines4[3].Param := 0; // G1 Continuous [Op37 P1]
    Lines4[4].X := 264.608; Lines4[4].Z := 267.140; Lines4[4].F := 1500; Lines4[4].CMD := 2; Lines4[4].Param := 0; // G1 Continuous [Op37 P1]
    Lines4[5].X := 268.845; Lines4[5].Z := 248.118; Lines4[5].F := 1500; Lines4[5].CMD := 2; Lines4[5].Param := 0; // G1 Continuous [Op37 P1]
    Lines4[6].X := 272.169; Lines4[6].Z := 181.000; Lines4[6].F := 0; Lines4[6].CMD := 0; Lines4[6].Param := 0; // G0 Rapid [Op38 P1]
    Lines4[7].X := 273.320; Lines4[7].Z := 206.779; Lines4[7].F := 1500; Lines4[7].CMD := 2; Lines4[7].Param := 0; // G1 Continuous [Op38 P1]
    Lines4[8].X := 271.668; Lines4[8].Z := 237.093; Lines4[8].F := 1500; Lines4[8].CMD := 2; Lines4[8].Param := 0; // G1 Continuous [Op38 P1]
    Lines4[9].X := 266.663; Lines4[9].Z := 267.119; Lines4[9].F := 1500; Lines4[9].CMD := 2; Lines4[9].Param := 0; // G1 Continuous [Op38 P1]
    Lines4[10].X := 258.243; Lines4[10].Z := 297.185; Lines4[10].F := 1500; Lines4[10].CMD := 2; Lines4[10].Param := 0; // G1 Continuous [Op38 P1]
    Lines4[11].X := 246.639; Lines4[11].Z := 326.346; Lines4[11].F := 1500; Lines4[11].CMD := 2; Lines4[11].Param := 0; // G1 Continuous [Op38 P1]
    Lines4[12].X := 224.375; Lines4[12].Z := 316.696; Lines4[12].F := 0; Lines4[12].CMD := 0; Lines4[12].Param := 0; // G0 Rapid [Op39 P1]
    Lines4[13].X := 235.640; Lines4[13].Z := 305.828; Lines4[13].F := 1500; Lines4[13].CMD := 2; Lines4[13].Param := 0; // G1 Continuous [Op39 P1]
    Lines4[14].X := 245.758; Lines4[14].Z := 294.025; Lines4[14].F := 1500; Lines4[14].CMD := 2; Lines4[14].Param := 0; // G1 Continuous [Op39 P1]
    Lines4[15].X := 254.384; Lines4[15].Z := 281.679; Lines4[15].F := 1500; Lines4[15].CMD := 2; Lines4[15].Param := 0; // G1 Continuous [Op39 P1]
    Lines4[16].X := 261.408; Lines4[16].Z := 268.991; Lines4[16].F := 1500; Lines4[16].CMD := 2; Lines4[16].Param := 0; // G1 Continuous [Op39 P1]
    Lines4[17].X := 266.677; Lines4[17].Z := 256.373; Lines4[17].F := 1500; Lines4[17].CMD := 2; Lines4[17].Param := 0; // G1 Continuous [Op39 P1]
    Lines4[18].X := 270.363; Lines4[18].Z := 243.511; Lines4[18].F := 1500; Lines4[18].CMD := 2; Lines4[18].Param := 0; // G1 Continuous [Op39 P1]
    Lines4[19].X := 272.557; Lines4[19].Z := 230.042; Lines4[19].F := 1500; Lines4[19].CMD := 2; Lines4[19].Param := 0; // G1 Continuous [Op39 P1]
    Lines4[20].X := 273.291; Lines4[20].Z := 215.866; Lines4[20].F := 1500; Lines4[20].CMD := 2; Lines4[20].Param := 0; // G1 Continuous [Op39 P1]
    Lines4[21].X := 272.270; Lines4[21].Z := 198.643; Lines4[21].F := 1500; Lines4[21].CMD := 2; Lines4[21].Param := 0; // G1 Continuous [Op39 P1]
    Lines4[22].X := 269.221; Lines4[22].Z := 181.000; Lines4[22].F := 1500; Lines4[22].CMD := 1; Lines4[22].Param := 0; // G1 Linear [Op39 P1]
    Lines4[23].X := 270.721; Lines4[23].Z := 181.000; Lines4[23].F := 1500; Lines4[23].CMD := 1; Lines4[23].Param := 0; // G1 Linear [Op40 P1]
    Lines4[24].X := 272.649; Lines4[24].Z := 197.967; Lines4[24].F := 1500; Lines4[24].CMD := 2; Lines4[24].Param := 0; // G1 Continuous [Op40 P1]
    Lines4[25].X := 273.294; Lines4[25].Z := 214.819; Lines4[25].F := 1500; Lines4[25].CMD := 2; Lines4[25].Param := 0; // G1 Continuous [Op40 P1]
    Lines4[26].X := 271.378; Lines4[26].Z := 243.212; Lines4[26].F := 1500; Lines4[26].CMD := 2; Lines4[26].Param := 0; // G1 Continuous [Op40 P1]
    Lines4[27].X := 265.628; Lines4[27].Z := 270.594; Lines4[27].F := 1500; Lines4[27].CMD := 2; Lines4[27].Param := 0; // G1 Continuous [Op40 P1]
    Lines4[28].X := 255.766; Lines4[28].Z := 298.151; Lines4[28].F := 1500; Lines4[28].CMD := 2; Lines4[28].Param := 0; // G1 Continuous [Op40 P1]
    Lines4[29].X := 242.197; Lines4[29].Z := 324.548; Lines4[29].F := 1500; Lines4[29].CMD := 1; Lines4[29].Param := 0; // G1 Linear [Op40 P1]
    Lines4[30].X := 251.208; Lines4[30].Z := 307.990; Lines4[30].F := 1500; Lines4[30].CMD := 2; Lines4[30].Param := 0; // G1 Continuous [Op40 P1]
    Lines4[31].X := 258.852; Lines4[31].Z := 290.686; Lines4[31].F := 1500; Lines4[31].CMD := 2; Lines4[31].Param := 0; // G1 Continuous [Op40 P1]
    Lines4[32].X := 264.854; Lines4[32].Z := 273.261; Lines4[32].F := 1500; Lines4[32].CMD := 2; Lines4[32].Param := 0; // G1 Continuous [Op40 P1]
    Lines4[33].X := 269.269; Lines4[33].Z := 255.604; Lines4[33].F := 1500; Lines4[33].CMD := 1; Lines4[33].Param := 0; // G1 Linear [Op40 P1]
    Lines4[34].X := 260.885; Lines4[34].Z := 289.121; Lines4[34].F := 1500; Lines4[34].CMD := 2; Lines4[34].Param := 0; // G1 Continuous [Op41 P1]
    Lines4[35].X := 248.040; Lines4[35].Z := 321.829; Lines4[35].F := 1500; Lines4[35].CMD := 1; Lines4[35].Param := 0; // G1 Linear [Op41 P1]
    Lines4[36].X := 255.433; Lines4[36].Z := 304.528; Lines4[36].F := 1500; Lines4[36].CMD := 2; Lines4[36].Param := 0; // G1 Continuous [Op41 P1]
    Lines4[37].X := 261.567; Lines4[37].Z := 286.962; Lines4[37].F := 1500; Lines4[37].CMD := 2; Lines4[37].Param := 0; // G1 Continuous [Op41 P1]
    Lines4[38].X := 266.421; Lines4[38].Z := 269.245; Lines4[38].F := 1500; Lines4[38].CMD := 2; Lines4[38].Param := 0; // G1 Continuous [Op41 P1]
    Lines4[39].X := 269.997; Lines4[39].Z := 251.369; Lines4[39].F := 1500; Lines4[39].CMD := 2; Lines4[39].Param := 0; // G1 Continuous [Op41 P1]
    Lines4[40].X := 271.350; Lines4[40].Z := 181.000; Lines4[40].F := 0; Lines4[40].CMD := 0; Lines4[40].Param := 0; // G0 Rapid [Op42 P1]
    Lines4[41].X := 273.295; Lines4[41].Z := 214.285; Lines4[41].F := 1500; Lines4[41].CMD := 2; Lines4[41].Param := 0; // G1 Continuous [Op42 P1]
    Lines4[42].X := 271.831; Lines4[42].Z := 242.875; Lines4[42].F := 1500; Lines4[42].CMD := 2; Lines4[42].Param := 0; // G1 Continuous [Op42 P1]
    Lines4[43].X := 267.409; Lines4[43].Z := 270.928; Lines4[43].F := 1500; Lines4[43].CMD := 2; Lines4[43].Param := 0; // G1 Continuous [Op42 P1]
    Lines4[44].X := 259.903; Lines4[44].Z := 299.103; Lines4[44].F := 1500; Lines4[44].CMD := 2; Lines4[44].Param := 0; // G1 Continuous [Op42 P1]
    Lines4[45].X := 249.512; Lines4[45].Z := 326.552; Lines4[45].F := 1500; Lines4[45].CMD := 2; Lines4[45].Param := 0; // G1 Continuous [Op42 P1]
    Lines4[46].X := 227.898; Lines4[46].Z := 323.233; Lines4[46].F := 0; Lines4[46].CMD := 0; Lines4[46].Param := 0; // G0 Rapid [Op43 P1]
    Lines4[47].X := 238.460; Lines4[47].Z := 312.413; Lines4[47].F := 1500; Lines4[47].CMD := 2; Lines4[47].Param := 0; // G1 Continuous [Op43 P1]
    Lines4[48].X := 247.897; Lines4[48].Z := 300.794; Lines4[48].F := 1500; Lines4[48].CMD := 2; Lines4[48].Param := 0; // G1 Continuous [Op43 P1]
    Lines4[49].X := 255.891; Lines4[49].Z := 288.733; Lines4[49].F := 1500; Lines4[49].CMD := 2; Lines4[49].Param := 0; // G1 Continuous [Op43 P1]
    Lines4[50].X := 262.347; Lines4[50].Z := 276.397; Lines4[50].F := 1500; Lines4[50].CMD := 2; Lines4[50].Param := 0; // G1 Continuous [Op43 P1]
    Lines4[51].X := 267.134; Lines4[51].Z := 264.171; Lines4[51].F := 1500; Lines4[51].CMD := 2; Lines4[51].Param := 0; // G1 Continuous [Op43 P1]
    Lines4[52].X := 270.511; Lines4[52].Z := 251.476; Lines4[52].F := 1500; Lines4[52].CMD := 2; Lines4[52].Param := 0; // G1 Continuous [Op43 P1]
    Lines4[53].X := 272.573; Lines4[53].Z := 237.938; Lines4[53].F := 1500; Lines4[53].CMD := 2; Lines4[53].Param := 0; // G1 Continuous [Op43 P1]
    Lines4[54].X := 273.264; Lines4[54].Z := 223.690; Lines4[54].F := 1500; Lines4[54].CMD := 2; Lines4[54].Param := 0; // G1 Continuous [Op43 P1]
    Lines4[55].X := 271.811; Lines4[55].Z := 202.568; Lines4[55].F := 1500; Lines4[55].CMD := 2; Lines4[55].Param := 0; // G1 Continuous [Op43 P1]
    Lines4[56].X := 267.466; Lines4[56].Z := 181.000; Lines4[56].F := 1500; Lines4[56].CMD := 1; Lines4[56].Param := 0; // G1 Linear [Op43 P1]
    Lines4[57].X := 270.242; Lines4[57].Z := 181.000; Lines4[57].F := 1500; Lines4[57].CMD := 1; Lines4[57].Param := 0; // G1 Linear [Op44 P1]
    Lines4[58].X := 272.505; Lines4[58].Z := 201.448; Lines4[58].F := 1500; Lines4[58].CMD := 2; Lines4[58].Param := 0; // G1 Continuous [Op44 P1]
    Lines4[59].X := 273.270; Lines4[59].Z := 222.054; Lines4[59].F := 1500; Lines4[59].CMD := 2; Lines4[59].Param := 0; // G1 Continuous [Op44 P1]
    Lines4[60].X := 271.800; Lines4[60].Z := 250.193; Lines4[60].F := 1500; Lines4[60].CMD := 2; Lines4[60].Param := 0; // G1 Continuous [Op44 P1]
    Lines4[61].X := 267.423; Lines4[61].Z := 277.502; Lines4[61].F := 1500; Lines4[61].CMD := 2; Lines4[61].Param := 0; // G1 Continuous [Op44 P1]
    Lines4[62].X := 259.957; Lines4[62].Z := 304.891; Lines4[62].F := 1500; Lines4[62].CMD := 2; Lines4[62].Param := 0; // G1 Continuous [Op44 P1]
    Lines4[63].X := 249.623; Lines4[63].Z := 331.547; Lines4[63].F := 1500; Lines4[63].CMD := 1; Lines4[63].Param := 0; // G1 Linear [Op44 P1]
    Lines4[64].X := 257.157; Lines4[64].Z := 312.957; Lines4[64].F := 1500; Lines4[64].CMD := 2; Lines4[64].Param := 0; // G1 Continuous [Op44 P1]
    Lines4[65].X := 263.276; Lines4[65].Z := 294.083; Lines4[65].F := 1500; Lines4[65].CMD := 2; Lines4[65].Param := 0; // G1 Continuous [Op44 P1]
    Lines4[66].X := 267.942; Lines4[66].Z := 275.041; Lines4[66].F := 1500; Lines4[66].CMD := 2; Lines4[66].Param := 0; // G1 Continuous [Op44 P1]
    Lines4[67].X := 271.151; Lines4[67].Z := 255.763; Lines4[67].F := 1500; Lines4[67].CMD := 1; Lines4[67].Param := 0; // G1 Linear [Op44 P1]
    Lines4[68].X := 264.213; Lines4[68].Z := 293.130; Lines4[68].F := 1500; Lines4[68].CMD := 2; Lines4[68].Param := 0; // G1 Continuous [Op45 P1]
    Lines4[69].X := 252.358; Lines4[69].Z := 330.185; Lines4[69].F := 1500; Lines4[69].CMD := 1; Lines4[69].Param := 0; // G1 Linear [Op45 P1]
    Lines4[70].X := 264.396; Lines4[70].Z := 292.398; Lines4[70].F := 1500; Lines4[70].CMD := 2; Lines4[70].Param := 0; // G1 Continuous [Op45 P1]
    Lines4[71].X := 268.526; Lines4[71].Z := 273.223; Lines4[71].F := 1500; Lines4[71].CMD := 2; Lines4[71].Param := 0; // G1 Continuous [Op45 P1]
    Lines4[72].X := 271.374; Lines4[72].Z := 253.852; Lines4[72].F := 1500; Lines4[72].CMD := 2; Lines4[72].Param := 0; // G1 Continuous [Op45 P1]
    Lines4[73].X := 270.789; Lines4[73].Z := 181.000; Lines4[73].F := 0; Lines4[73].CMD := 0; Lines4[73].Param := 0; // G0 Rapid [Op46 P1]
    Lines4[74].X := 273.270; Lines4[74].Z := 221.597; Lines4[74].F := 1500; Lines4[74].CMD := 2; Lines4[74].Param := 0; // G1 Continuous [Op46 P1]
    Lines4[75].X := 272.069; Lines4[75].Z := 249.738; Lines4[75].F := 1500; Lines4[75].CMD := 2; Lines4[75].Param := 0; // G1 Continuous [Op46 P1]
    Lines4[76].X := 268.446; Lines4[76].Z := 277.408; Lines4[76].F := 1500; Lines4[76].CMD := 2; Lines4[76].Param := 0; // G1 Continuous [Op46 P1]
    Lines4[77].X := 262.301; Lines4[77].Z := 305.125; Lines4[77].F := 1500; Lines4[77].CMD := 2; Lines4[77].Param := 0; // G1 Continuous [Op46 P1]
    Lines4[78].X := 253.731; Lines4[78].Z := 332.415; Lines4[78].F := 1500; Lines4[78].CMD := 2; Lines4[78].Param := 0; // G1 Continuous [Op46 P1]
    Lines4[79].X := 235.424; Lines4[79].Z := 326.307; Lines4[79].F := 0; Lines4[79].CMD := 0; Lines4[79].Param := 0; // G0 Rapid [Op47 P1]
    Lines4[80].X := 252.307; Lines4[80].Z := 305.657; Lines4[80].F := 1500; Lines4[80].CMD := 2; Lines4[80].Param := 0; // G1 Continuous [Op47 P1]
    Lines4[81].X := 258.866; Lines4[81].Z := 294.890; Lines4[81].F := 1500; Lines4[81].CMD := 2; Lines4[81].Param := 0; // G1 Continuous [Op47 P1]
    Lines4[82].X := 264.070; Lines4[82].Z := 283.978; Lines4[82].F := 1500; Lines4[82].CMD := 2; Lines4[82].Param := 0; // G1 Continuous [Op47 P1]
    Lines4[83].X := 268.069; Lines4[83].Z := 272.544; Lines4[83].F := 1500; Lines4[83].CMD := 2; Lines4[83].Param := 0; // G1 Continuous [Op47 P1]
    Lines4[84].X := 270.932; Lines4[84].Z := 260.444; Lines4[84].F := 1500; Lines4[84].CMD := 2; Lines4[84].Param := 0; // G1 Continuous [Op47 P1]
    Lines4[85].X := 273.228; Lines4[85].Z := 234.672; Lines4[85].F := 1500; Lines4[85].CMD := 2; Lines4[85].Param := 0; // G1 Continuous [Op47 P1]
    Lines4[86].X := 270.979; Lines4[86].Z := 207.681; Lines4[86].F := 1500; Lines4[86].CMD := 2; Lines4[86].Param := 0; // G1 Continuous [Op47 P1]
    Lines4[87].X := 264.404; Lines4[87].Z := 181.001; Lines4[87].F := 1500; Lines4[87].CMD := 1; Lines4[87].Param := 0; // G1 Linear [Op47 P1]
    Lines4[88].X := 269.664; Lines4[88].Z := 181.001; Lines4[88].F := 1500; Lines4[88].CMD := 1; Lines4[88].Param := 0; // G1 Linear [Op48 P1]
    Lines4[89].X := 272.353; Lines4[89].Z := 205.217; Lines4[89].F := 1500; Lines4[89].CMD := 2; Lines4[89].Param := 0; // G1 Continuous [Op48 P1]
    Lines4[90].X := 273.245; Lines4[90].Z := 229.375; Lines4[90].F := 1500; Lines4[90].CMD := 2; Lines4[90].Param := 0; // G1 Continuous [Op48 P1]
    Lines4[91].X := 272.152; Lines4[91].Z := 255.805; Lines4[91].F := 1500; Lines4[91].CMD := 2; Lines4[91].Param := 0; // G1 Continuous [Op48 P1]
    Lines4[92].X := 268.882; Lines4[92].Z := 281.766; Lines4[92].F := 1500; Lines4[92].CMD := 2; Lines4[92].Param := 0; // G1 Continuous [Op48 P1]
    Lines4[93].X := 263.421; Lines4[93].Z := 307.306; Lines4[93].F := 1500; Lines4[93].CMD := 2; Lines4[93].Param := 0; // G1 Continuous [Op48 P1]
    Lines4[94].X := 255.724; Lines4[94].Z := 332.753; Lines4[94].F := 1500; Lines4[94].CMD := 1; Lines4[94].Param := 0; // G1 Linear [Op48 P1]
    Lines4[95].X := 266.472; Lines4[95].Z := 294.353; Lines4[95].F := 1500; Lines4[95].CMD := 2; Lines4[95].Param := 0; // G1 Continuous [Op48 P1]
    Lines4[96].X := 272.153; Lines4[96].Z := 255.794; Lines4[96].F := 1500; Lines4[96].CMD := 1; Lines4[96].Param := 0; // G1 Linear [Op48 P1]
    Lines4[97].X := 267.125; Lines4[97].Z := 294.687; Lines4[97].F := 1500; Lines4[97].CMD := 2; Lines4[97].Param := 0; // G1 Continuous [Op49 P1]
    Lines4[98].X := 257.883; Lines4[98].Z := 333.451; Lines4[98].F := 1500; Lines4[98].CMD := 1; Lines4[98].Param := 0; // G1 Linear [Op49 P1]
    Lines4[99].X := 267.527; Lines4[99].Z := 292.465; Lines4[99].F := 1500; Lines4[99].CMD := 2; Lines4[99].Param := 0; // G1 Continuous [Op49 P1]

    // --- Lines5 (global lines 400..499) ---
    Lines5[0].X := 272.475; Lines5[0].Z := 251.168; Lines5[0].F := 1500; Lines5[0].CMD := 2; Lines5[0].Param := 0; // G1 Continuous [Op49 P1]
    Lines5[1].X := 269.782; Lines5[1].Z := 181.001; Lines5[1].F := 0; Lines5[1].CMD := 0; Lines5[1].Param := 0; // G0 Rapid [Op50 P1]
    Lines5[2].X := 272.367; Lines5[2].Z := 206.221; Lines5[2].F := 1500; Lines5[2].CMD := 2; Lines5[2].Param := 0; // G1 Continuous [Op50 P1]
    Lines5[3].X := 273.237; Lines5[3].Z := 231.614; Lines5[3].F := 1500; Lines5[3].CMD := 2; Lines5[3].Param := 0; // G1 Continuous [Op50 P1]
    Lines5[4].X := 272.321; Lines5[4].Z := 257.519; Lines5[4].F := 1500; Lines5[4].CMD := 2; Lines5[4].Param := 0; // G1 Continuous [Op50 P1]
    Lines5[5].X := 269.583; Lines5[5].Z := 283.015; Lines5[5].F := 1500; Lines5[5].CMD := 2; Lines5[5].Param := 0; // G1 Continuous [Op50 P1]
    Lines5[6].X := 265.007; Lines5[6].Z := 308.197; Lines5[6].F := 1500; Lines5[6].CMD := 2; Lines5[6].Param := 0; // G1 Continuous [Op50 P1]
    Lines5[7].X := 258.593; Lines5[7].Z := 333.205; Lines5[7].F := 1500; Lines5[7].CMD := 2; Lines5[7].Param := 0; // G1 Continuous [Op50 P1]
    Lines5[8].X := 244.286; Lines5[8].Z := 325.150; Lines5[8].F := 0; Lines5[8].CMD := 0; Lines5[8].Param := 0; // G0 Rapid [Op51 P1]
    Lines5[9].X := 257.290; Lines5[9].Z := 307.939; Lines5[9].F := 1372; Lines5[9].CMD := 2; Lines5[9].Param := 0; // G1 Continuous [Op51 P1]
    Lines5[10].X := 265.942; Lines5[10].Z := 290.097; Lines5[10].F := 1359; Lines5[10].CMD := 2; Lines5[10].Param := 0; // G1 Continuous [Op51 P1]
    Lines5[11].X := 271.386; Lines5[11].Z := 269.136; Lines5[11].F := 1359; Lines5[11].CMD := 2; Lines5[11].Param := 0; // G1 Continuous [Op51 P1]
    Lines5[12].X := 273.189; Lines5[12].Z := 246.305; Lines5[12].F := 1500; Lines5[12].CMD := 2; Lines5[12].Param := 0; // G1 Continuous [Op51 P1]
    Lines5[13].X := 272.340; Lines5[13].Z := 229.985; Lines5[13].F := 1500; Lines5[13].CMD := 2; Lines5[13].Param := 0; // G1 Continuous [Op51 P1]
    Lines5[14].X := 269.802; Lines5[14].Z := 213.296; Lines5[14].F := 1500; Lines5[14].CMD := 2; Lines5[14].Param := 0; // G1 Continuous [Op51 P1]
    Lines5[15].X := 265.661; Lines5[15].Z := 196.843; Lines5[15].F := 1500; Lines5[15].CMD := 2; Lines5[15].Param := 0; // G1 Continuous [Op51 P1]
    Lines5[16].X := 260.014; Lines5[16].Z := 181.001; Lines5[16].F := 1500; Lines5[16].CMD := 1; Lines5[16].Param := 0; // G1 Linear [Op51 P1]
    Lines5[17].X := 266.490; Lines5[17].Z := 181.001; Lines5[17].F := 1500; Lines5[17].CMD := 1; Lines5[17].Param := 0; // G1 Linear [Op52 P1]
    Lines5[18].X := 271.514; Lines5[18].Z := 212.848; Lines5[18].F := 1500; Lines5[18].CMD := 2; Lines5[18].Param := 0; // G1 Continuous [Op52 P1]
    Lines5[19].X := 273.193; Lines5[19].Z := 244.972; Lines5[19].F := 1500; Lines5[19].CMD := 2; Lines5[19].Param := 0; // G1 Continuous [Op52 P1]
    Lines5[20].X := 272.298; Lines5[20].Z := 268.012; Lines5[20].F := 1500; Lines5[20].CMD := 2; Lines5[20].Param := 0; // G1 Continuous [Op52 P1]
    Lines5[21].X := 269.675; Lines5[21].Z := 290.349; Lines5[21].F := 1500; Lines5[21].CMD := 2; Lines5[21].Param := 0; // G1 Continuous [Op52 P1]
    Lines5[22].X := 265.398; Lines5[22].Z := 311.817; Lines5[22].F := 1500; Lines5[22].CMD := 2; Lines5[22].Param := 0; // G1 Continuous [Op52 P1]
    Lines5[23].X := 259.211; Lines5[23].Z := 333.518; Lines5[23].F := 1500; Lines5[23].CMD := 1; Lines5[23].Param := 0; // G1 Linear [Op52 P1]
    Lines5[24].X := 264.796; Lines5[24].Z := 314.254; Lines5[24].F := 1500; Lines5[24].CMD := 2; Lines5[24].Param := 0; // G1 Continuous [Op52 P1]
    Lines5[25].X := 268.843; Lines5[25].Z := 295.323; Lines5[25].F := 1500; Lines5[25].CMD := 2; Lines5[25].Param := 0; // G1 Continuous [Op52 P1]
    Lines5[26].X := 271.609; Lines5[26].Z := 275.572; Lines5[26].F := 1500; Lines5[26].CMD := 2; Lines5[26].Param := 0; // G1 Continuous [Op52 P1]
    Lines5[27].X := 273.004; Lines5[27].Z := 255.531; Lines5[27].F := 1500; Lines5[27].CMD := 1; Lines5[27].Param := 0; // G1 Linear [Op52 P1]
    Lines5[28].X := 269.237; Lines5[28].Z := 294.216; Lines5[28].F := 1500; Lines5[28].CMD := 2; Lines5[28].Param := 0; // G1 Continuous [Op53 P1]
    Lines5[29].X := 260.705; Lines5[29].Z := 331.131; Lines5[29].F := 1500; Lines5[29].CMD := 1; Lines5[29].Param := 0; // G1 Linear [Op53 P1]
    Lines5[30].X := 265.765; Lines5[30].Z := 311.986; Lines5[30].F := 1500; Lines5[30].CMD := 2; Lines5[30].Param := 0; // G1 Continuous [Op53 P1]
    Lines5[31].X := 269.437; Lines5[31].Z := 292.972; Lines5[31].F := 1500; Lines5[31].CMD := 2; Lines5[31].Param := 0; // G1 Continuous [Op53 P1]
    Lines5[32].X := 271.902; Lines5[32].Z := 273.181; Lines5[32].F := 1500; Lines5[32].CMD := 2; Lines5[32].Param := 0; // G1 Continuous [Op53 P1]
    Lines5[33].X := 273.083; Lines5[33].Z := 252.924; Lines5[33].F := 1500; Lines5[33].CMD := 2; Lines5[33].Param := 0; // G1 Continuous [Op53 P1]
    Lines5[34].X := 266.869; Lines5[34].Z := 181.001; Lines5[34].F := 0; Lines5[34].CMD := 0; Lines5[34].Param := 0; // G0 Rapid [Op54 P1]
    Lines5[35].X := 271.595; Lines5[35].Z := 213.863; Lines5[35].F := 1500; Lines5[35].CMD := 2; Lines5[35].Param := 0; // G1 Continuous [Op54 P1]
    Lines5[36].X := 273.186; Lines5[36].Z := 247.180; Lines5[36].F := 1500; Lines5[36].CMD := 2; Lines5[36].Param := 0; // G1 Continuous [Op54 P1]
    Lines5[37].X := 272.488; Lines5[37].Z := 268.911; Lines5[37].F := 1500; Lines5[37].CMD := 2; Lines5[37].Param := 0; // G1 Continuous [Op54 P1]
    Lines5[38].X := 270.423; Lines5[38].Z := 290.259; Lines5[38].F := 1500; Lines5[38].CMD := 2; Lines5[38].Param := 0; // G1 Continuous [Op54 P1]
    Lines5[39].X := 267.013; Lines5[39].Z := 311.107; Lines5[39].F := 1500; Lines5[39].CMD := 2; Lines5[39].Param := 0; // G1 Continuous [Op54 P1]
    Lines5[40].X := 262.172; Lines5[40].Z := 331.852; Lines5[40].F := 1500; Lines5[40].CMD := 2; Lines5[40].Param := 0; // G1 Continuous [Op54 P1]
    Lines5[41].X := 273.391; Lines5[41].Z := 181.001; Lines5[41].F := 0; Lines5[41].CMD := 0; Lines5[41].Param := 0; // G0 Rapid [Op55 P1]
    Lines5[42].X := 273.050; Lines5[42].Z := 283.412; Lines5[42].F := 1389; Lines5[42].CMD := 2; Lines5[42].Param := 0; // G1 Continuous [Op55 P1]
    Lines5[43].X := 272.825; Lines5[43].Z := 284.543; Lines5[43].F := 1389; Lines5[43].CMD := 2; Lines5[43].Param := 0; // G1 Continuous [Op55 P1]
    Lines5[44].X := 264.337; Lines5[44].Z := 310.391; Lines5[44].F := 770; Lines5[44].CMD := 2; Lines5[44].Param := 0; // G1 Continuous [Op55 P1]
    Lines5[45].X := 259.181; Lines5[45].Z := 316.888; Lines5[45].F := 770; Lines5[45].CMD := 2; Lines5[45].Param := 0; // G1 Continuous [Op55 P1]
    Lines5[46].X := 250.803; Lines5[46].Z := 322.123; Lines5[46].F := 796; Lines5[46].CMD := 1; Lines5[46].Param := 0; // G1 Linear [Op55 P1]
    Lines5[47].X := 259.181; Lines5[47].Z := 316.888; Lines5[47].F := 796; Lines5[47].CMD := 2; Lines5[47].Param := 0; // G1 Continuous [Op55 P1]
    Lines5[48].X := 264.337; Lines5[48].Z := 310.391; Lines5[48].F := 760; Lines5[48].CMD := 2; Lines5[48].Param := 0; // G1 Continuous [Op55 P1]
    Lines5[49].X := 273.050; Lines5[49].Z := 283.412; Lines5[49].F := 760; Lines5[49].CMD := 2; Lines5[49].Param := 0; // G1 Continuous [Op55 P1]
    Lines5[50].X := 255.430; Lines5[50].Z := 318.457; Lines5[50].F := 0; Lines5[50].CMD := 0; Lines5[50].Param := 0; // G0 Rapid [Op56 P1]
    Lines5[51].X := 262.281; Lines5[51].Z := 314.748; Lines5[51].F := 707; Lines5[51].CMD := 2; Lines5[51].Param := 0; // G1 Continuous [Op56 P1]
    Lines5[52].X := 266.352; Lines5[52].Z := 309.794; Lines5[52].F := 707; Lines5[52].CMD := 2; Lines5[52].Param := 0; // G1 Continuous [Op56 P1]
    Lines5[53].X := 272.794; Lines5[53].Z := 289.557; Lines5[53].F := 719; Lines5[53].CMD := 2; Lines5[53].Param := 0; // G1 Continuous [Op56 P1]
    Lines5[54].X := 273.033; Lines5[54].Z := 288.394; Lines5[54].F := 1346; Lines5[54].CMD := 2; Lines5[54].Param := 0; // G1 Continuous [Op56 P1]
    Lines5[55].X := 273.141; Lines5[55].Z := 256.000; Lines5[55].F := 1346; Lines5[55].CMD := 2; Lines5[55].Param := 0; // G1 Continuous [Op56 P1]
    Lines5[56].X := 273.391; Lines5[56].Z := 181.001; Lines5[56].F := 0; Lines5[56].CMD := 0; Lines5[56].Param := 0; // G0 Rapid [Op57 P1]
    Lines5[57].X := 273.033; Lines5[57].Z := 288.359; Lines5[57].F := 1276; Lines5[57].CMD := 2; Lines5[57].Param := 0; // G1 Continuous [Op57 P1]
    Lines5[58].X := 272.767; Lines5[58].Z := 289.584; Lines5[58].F := 1276; Lines5[58].CMD := 2; Lines5[58].Param := 0; // G1 Continuous [Op57 P1]
    Lines5[59].X := 263.396; Lines5[59].Z := 315.132; Lines5[59].F := 769; Lines5[59].CMD := 2; Lines5[59].Param := 0; // G1 Continuous [Op57 P1]
    Lines5[60].X := 258.018; Lines5[60].Z := 321.449; Lines5[60].F := 769; Lines5[60].CMD := 2; Lines5[60].Param := 0; // G1 Continuous [Op57 P1]
    Lines5[61].X := 249.464; Lines5[61].Z := 326.395; Lines5[61].F := 796; Lines5[61].CMD := 2; Lines5[61].Param := 0; // G1 Continuous [Op57 P1]
    Lines5[62].X := 273.391; Lines5[62].Z := 181.001; Lines5[62].F := 0; Lines5[62].CMD := 0; Lines5[62].Param := 0; // G0 Rapid [Op58 P1]
    Lines5[63].X := 273.017; Lines5[63].Z := 293.141; Lines5[63].F := 968; Lines5[63].CMD := 2; Lines5[63].Param := 0; // G1 Continuous [Op58 P1]
    Lines5[64].X := 272.557; Lines5[64].Z := 294.727; Lines5[64].F := 968; Lines5[64].CMD := 2; Lines5[64].Param := 0; // G1 Continuous [Op58 P1]
    Lines5[65].X := 259.781; Lines5[65].Z := 318.773; Lines5[65].F := 770; Lines5[65].CMD := 2; Lines5[65].Param := 0; // G1 Continuous [Op58 P1]
    Lines5[66].X := 253.589; Lines5[66].Z := 324.301; Lines5[66].F := 770; Lines5[66].CMD := 2; Lines5[66].Param := 0; // G1 Continuous [Op58 P1]
    Lines5[67].X := 244.435; Lines5[67].Z := 328.039; Lines5[67].F := 797; Lines5[67].CMD := 2; Lines5[67].Param := 0; // G1 Continuous [Op58 P1]
    Lines5[68].X := 273.391; Lines5[68].Z := 181.001; Lines5[68].F := 0; Lines5[68].CMD := 0; Lines5[68].Param := 0; // G0 Rapid [Op59 P1]
    Lines5[69].X := 273.001; Lines5[69].Z := 298.135; Lines5[69].F := 962; Lines5[69].CMD := 2; Lines5[69].Param := 0; // G1 Continuous [Op59 P1]
    Lines5[70].X := 272.535; Lines5[70].Z := 299.731; Lines5[70].F := 962; Lines5[70].CMD := 2; Lines5[70].Param := 0; // G1 Continuous [Op59 P1]
    Lines5[71].X := 259.702; Lines5[71].Z := 323.678; Lines5[71].F := 770; Lines5[71].CMD := 2; Lines5[71].Param := 0; // G1 Continuous [Op59 P1]
    Lines5[72].X := 253.331; Lines5[72].Z := 329.325; Lines5[72].F := 770; Lines5[72].CMD := 2; Lines5[72].Param := 0; // G1 Continuous [Op59 P1]
    Lines5[73].X := 244.210; Lines5[73].Z := 333.005; Lines5[73].F := 795; Lines5[73].CMD := 2; Lines5[73].Param := 0; // G1 Continuous [Op59 P1]
    Lines5[74].X := 244.210; Lines5[74].Z := 333.005; Lines5[74].F := 0; Lines5[74].CMD := 20; Lines5[74].Param := 80; // Spindle ON 800 RPM [Op59 P1]
    Lines5[75].X := 273.391; Lines5[75].Z := 181.001; Lines5[75].F := 0; Lines5[75].CMD := 0; Lines5[75].Param := 0; // G0 Rapid [Op60 P1]
    Lines5[76].X := 272.984; Lines5[76].Z := 303.135; Lines5[76].F := 962; Lines5[76].CMD := 2; Lines5[76].Param := 0; // G1 Continuous [Op60 P1]
    Lines5[77].X := 272.518; Lines5[77].Z := 304.731; Lines5[77].F := 962; Lines5[77].CMD := 2; Lines5[77].Param := 0; // G1 Continuous [Op60 P1]
    Lines5[78].X := 259.685; Lines5[78].Z := 328.678; Lines5[78].F := 770; Lines5[78].CMD := 2; Lines5[78].Param := 0; // G1 Continuous [Op60 P1]
    Lines5[79].X := 253.315; Lines5[79].Z := 334.325; Lines5[79].F := 770; Lines5[79].CMD := 2; Lines5[79].Param := 0; // G1 Continuous [Op60 P1]
    Lines5[80].X := 244.193; Lines5[80].Z := 338.005; Lines5[80].F := 795; Lines5[80].CMD := 2; Lines5[80].Param := 0; // G1 Continuous [Op60 P1]
    Lines5[81].X := 273.391; Lines5[81].Z := 181.001; Lines5[81].F := 0; Lines5[81].CMD := 0; Lines5[81].Param := 0; // G0 Rapid [Op61 P1]
    Lines5[82].X := 272.968; Lines5[82].Z := 308.127; Lines5[82].F := 800; Lines5[82].CMD := 2; Lines5[82].Param := 0; // G1 Continuous [Op61 P1]
    Lines5[83].X := 272.494; Lines5[83].Z := 309.735; Lines5[83].F := 800; Lines5[83].CMD := 2; Lines5[83].Param := 0; // G1 Continuous [Op61 P1]
    Lines5[84].X := 261.156; Lines5[84].Z := 331.096; Lines5[84].F := 747; Lines5[84].CMD := 2; Lines5[84].Param := 0; // G1 Continuous [Op61 P1]
    Lines5[85].X := 255.453; Lines5[85].Z := 336.078; Lines5[85].F := 747; Lines5[85].CMD := 2; Lines5[85].Param := 0; // G1 Continuous [Op61 P1]
    Lines5[86].X := 247.215; Lines5[86].Z := 339.140; Lines5[86].F := 752; Lines5[86].CMD := 2; Lines5[86].Param := 0; // G1 Continuous [Op61 P1]
    Lines5[87].X := 217.215; Lines5[87].Z := 339.140; Lines5[87].F := 0; Lines5[87].CMD := 0; Lines5[87].Param := 0; // G0 Rapid [Op61 P1]
    Lines5[88].X := 273.391; Lines5[88].Z := 181.001; Lines5[88].F := 0; Lines5[88].CMD := 0; Lines5[88].Param := 0; // G0 Rapid [Op62 P1]
    Lines5[89].X := 272.951; Lines5[89].Z := 313.127; Lines5[89].F := 800; Lines5[89].CMD := 2; Lines5[89].Param := 0; // G1 Continuous [Op62 P1]
    Lines5[90].X := 272.477; Lines5[90].Z := 314.735; Lines5[90].F := 800; Lines5[90].CMD := 2; Lines5[90].Param := 0; // G1 Continuous [Op62 P1]
    Lines5[91].X := 261.139; Lines5[91].Z := 336.096; Lines5[91].F := 747; Lines5[91].CMD := 2; Lines5[91].Param := 0; // G1 Continuous [Op62 P1]
    Lines5[92].X := 255.436; Lines5[92].Z := 341.078; Lines5[92].F := 747; Lines5[92].CMD := 2; Lines5[92].Param := 0; // G1 Continuous [Op62 P1]
    Lines5[93].X := 247.199; Lines5[93].Z := 344.140; Lines5[93].F := 752; Lines5[93].CMD := 2; Lines5[93].Param := 0; // G1 Continuous [Op62 P1]
    Lines5[94].X := 217.199; Lines5[94].Z := 344.140; Lines5[94].F := 0; Lines5[94].CMD := 0; Lines5[94].Param := 0; // G0 Rapid [Op62 P1]
    Lines5[95].X := 217.199; Lines5[95].Z := 74.000; Lines5[95].F := 0; Lines5[95].CMD := 0; Lines5[95].Param := 0; // G0 Rapid [Op62 P1]
    Lines5[96].X := 174.000; Lines5[96].Z := 74.000; Lines5[96].F := 0; Lines5[96].CMD := 0; Lines5[96].Param := 0; // G0 Rapid [Op62 P1]
    Lines5[97].X := 174.000; Lines5[97].Z := 74.000; Lines5[97].F := 0; Lines5[97].CMD := 21; Lines5[97].Param := 0; // Spindle OFF [Op62 P1]
    Lines5[98].X := 174.000; Lines5[98].Z := 74.000; Lines5[98].F := 0; Lines5[98].CMD := 21; Lines5[98].Param := 0; // Spindle OFF
    Lines5[99].X := 0.000; Lines5[99].Z := 0.000; Lines5[99].F := 0; Lines5[99].CMD := 99; Lines5[99].Param := 0; // Program END
END_DATA_BLOCK